SPLINE
SPL {X  -134.058, Y  +288.094, Z    +0.000, E1   +46.503, E3 +177391.868}
SPL {X  -153.979, Y  +327.577, Z    +0.000, E1   +33.452, E3 +177403.408}
SPL {X  -160.130, Y  +351.024, Z    +0.000, E1   +21.715, E3 +177407.838}
SPL {X  -162.127, Y  +365.491, Z    +0.000, E1   +12.692, E3 +177407.762}
SPL {X  -162.801, Y  +378.004, Z    +0.000, E1    +3.811, E3 +177408.178}
SPL {X  -162.820, Y  +382.501, Z    +0.000, E1    +0.028, E3 +177407.596}
SPL {X  -162.820, Y  +385.123, Z    +0.000, E1    -3.284, E3 +177407.274}
SPL {X  -162.820, Y  +390.608, Z    +0.000, E1   -12.198, E3 +177407.187}
SPL {X  -162.820, Y  +396.028, Z    +0.000, E1   -22.022, E3 +177407.055}
SPL {X  -162.820, Y  +402.037, Z    +0.000, E1   -32.247, E3 +177406.993}
SPL {X  -162.820, Y  +411.189, Z    +0.000, E1   -44.140, E3 +177408.323}
SPL {X  -162.820, Y  +422.160, Z    +0.000, E1   -56.042, E3 +177406.794}
SPL {X  -162.820, Y  +475.891, Z    +0.000, E1   -67.666, E3 +177427.113}
SPL {X  -162.820, Y  +573.811, Z    +0.000, E1   -65.269, E3 +177511.711}
SPL {X  -162.820, Y  +580.233, Z    +0.000, E1   -64.427, E3 +177524.418}
SPL {X  -162.820, Y  +590.756, Z    +0.000, E1   -64.410, E3 +177534.986}
SPL {X  -162.820, Y  +600.605, Z    +0.000, E1   -64.446, E3 +177544.559}
SPL {X  -162.820, Y  +611.699, Z    +0.000, E1   -64.369, E3 +177556.238}
SPL {X  -162.820, Y  +622.825, Z    +0.000, E1   -64.446, E3 +177566.683}
SPL {X  -162.820, Y  +635.776, Z    +0.000, E1   -64.495, E3 +177579.372}
SPL {X  -162.820, Y  +648.933, Z    +0.000, E1   -64.417, E3 +177592.920}
SPL {X  -162.820, Y  +658.800, Z    +0.000, E1   -64.418, E3 +177602.734}
SPL {X  -162.820, Y  +670.777, Z    +0.000, E1   -64.432, E3 +177614.647}
SPL {X  -162.296, Y  +686.556, Z    +0.000, E1   -64.388, E3 +177630.850}
SPL {X  -160.469, Y  +701.070, Z    +0.000, E1   -64.058, E3 +177647.753}
SPL {X  -157.811, Y  +713.575, Z    +0.000, E1   -63.758, E3 +177662.332}
SPL {X  -154.601, Y  +724.576, Z    +0.000, E1   -63.303, E3 +177676.454}
SPL {X  -151.802, Y  +732.376, Z    +0.000, E1   -62.761, E3 +177687.581}
SPL {X  -149.758, Y  +737.398, Z    +0.000, E1   -62.434, E3 +177694.602}
SPL {X  -146.903, Y  +743.713, Z    +0.000, E1   -62.188, E3 +177702.375}
SPL {X  -144.901, Y  +747.758, Z    +0.000, E1   -61.566, E3 +177709.838}
SPL {X  -141.375, Y  +754.268, Z    +0.000, E1   -61.208, E3 +177718.391}
SPL {X  -137.988, Y  +759.927, Z    +0.000, E1   -60.537, E3 +177727.190}
SPL {X  -134.516, Y  +765.238, Z    +0.000, E1   -60.629, E3 +177731.993}
SPL {X  -126.113, Y  +776.485, Z    +0.000, E1   -62.672, E3 +177733.554}
SPL {X   -94.739, Y  +805.919, Z    +0.000, E1   -54.063, E3 +177840.294}
ENDSPLINE

SPLINE
SPL {X  -130.051, Y  +771.465, Z    +0.000, E1   -46.832, E3 +177962.078}
SPL {X  -150.288, Y  +736.141, Z    +0.000, E1   -36.889, E3 +177981.934}
SPL {X  -159.122, Y  +708.003, Z    +0.000, E1   -24.018, E3 +177984.643}
SPL {X  -161.938, Y  +690.423, Z    +0.000, E1   -13.625, E3 +177985.854}
SPL {X  -162.746, Y  +678.392, Z    +0.000, E1    -5.513, E3 +177985.927}
SPL {X  -162.820, Y  +672.097, Z    +0.000, E1    -0.584, E3 +177985.631}
SPL {X  -162.820, Y  +670.674, Z    +0.000, E1    +0.808, E3 +177985.263}
SPL {X  -162.820, Y  +666.307, Z    +0.000, E1    +6.851, E3 +177985.046}
SPL {X  -162.820, Y  +660.761, Z    +0.000, E1   +16.102, E3 +177985.188}
SPL {X  -162.820, Y  +655.024, Z    +0.000, E1   +25.730, E3 +177985.350}
SPL {X  -162.820, Y  +646.498, Z    +0.000, E1   +39.738, E3 +177983.871}
SPL {X  -162.820, Y  +637.711, Z    +0.000, E1   +46.793, E3 +177988.363}
SPL {X  -162.820, Y  +598.602, Z    +0.000, E1   +67.541, E3 +177990.914}
SPL {X  -162.820, Y  +578.435, Z    +0.000, E1   +65.472, E3 +178009.014}
SPL {X  -162.820, Y  +475.450, Z    +0.000, E1   +67.130, E3 +178077.952}
ENDSPLINE

SPLINE
SPL {X  -162.820, Y  +483.223, Z    +0.000, E1   +64.312, E3 +178092.391}
SPL {X  -162.820, Y  +502.830, Z    +0.000, E1   +59.229, E3 +178107.312}
ENDSPLINE

SPLINE
SPL {X  -162.820, Y  +486.621, Z    +0.000, E1   +59.661, E3 +178124.231}
SPL {X  -162.820, Y  +472.771, Z    +0.000, E1   +60.369, E3 +178135.977}
SPL {X  -162.820, Y  +460.138, Z    +0.000, E1   +61.014, E3 +178146.296}
SPL {X  -162.820, Y  +448.741, Z    +0.000, E1   +61.510, E3 +178155.811}
SPL {X  -162.820, Y  +430.985, Z    +0.000, E1   +62.533, E3 +178168.244}
SPL {X  -162.820, Y  +413.005, Z    +0.000, E1   +63.234, E3 +178182.234}
SPL {X  -162.820, Y  +396.727, Z    +0.000, E1   +63.972, E3 +178193.586}
SPL {X  -162.756, Y  +375.937, Z    +0.000, E1   +64.914, E3 +178207.195}
SPL {X  -161.353, Y  +358.691, Z    +0.000, E1   +65.588, E3 +178218.419}
SPL {X  -159.475, Y  +347.667, Z    +0.000, E1   +65.889, E3 +178226.300}
SPL {X  -157.043, Y  +337.513, Z    +0.000, E1   +65.541, E3 +178238.378}
SPL {X  -154.736, Y  +329.832, Z    +0.000, E1   +65.034, E3 +178248.824}
SPL {X  -151.631, Y  +321.184, Z    +0.000, E1   +64.776, E3 +178258.669}
SPL {X  -147.832, Y  +312.265, Z    +0.000, E1   +64.201, E3 +178270.478}
SPL {X  -145.264, Y  +306.955, Z    +0.000, E1   +63.555, E3 +178279.084}
SPL {X  -142.454, Y  +301.650, Z    +0.000, E1   +63.360, E3 +178285.088}
SPL {X  -139.696, Y  +296.861, Z    +0.000, E1   +62.910, E3 +178291.856}
SPL {X  -137.330, Y  +293.030, Z    +0.000, E1   +62.290, E3 +178298.481}
SPL {X  -134.245, Y  +288.366, Z    +0.000, E1   +62.031, E3 +178303.962}
SPL {X  -128.642, Y  +280.693, Z    +0.000, E1   +63.351, E3 +178304.956}
SPL {X   -90.696, Y  +245.280, Z    +0.000, E1   +54.124, E3 +178425.644}
ENDSPLINE

SPLINE
SPL {X  -134.058, Y  +288.094, Z    +0.000, E1   +46.503, E3 +178553.158}
SPL {X  -148.633, Y  +314.028, Z    +0.000, E1   +38.752, E3 +178562.047}
SPL {X  -156.325, Y  +334.971, Z    +0.000, E1   +30.037, E3 +178565.814}
SPL {X  -160.130, Y  +351.024, Z    +0.000, E1   +21.715, E3 +178569.128}
SPL {X  -162.127, Y  +365.491, Z    +0.000, E1   +12.692, E3 +178569.052}
SPL {X  -162.801, Y  +378.004, Z    +0.000, E1    +3.811, E3 +178569.468}
SPL {X  -162.820, Y  +382.997, Z    +0.000, E1    -0.389, E3 +178568.792}
SPL {X  -162.820, Y  +387.631, Z    +0.000, E1    -7.169, E3 +178568.551}
SPL {X  -162.820, Y  +394.064, Z    +0.000, E1   -18.298, E3 +178568.361}
SPL {X  -162.820, Y  +402.037, Z    +0.000, E1   -32.247, E3 +178568.283}
SPL {X  -162.820, Y  +414.067, Z    +0.000, E1   -47.235, E3 +178569.709}
SPL {X  -162.820, Y  +424.566, Z    +0.000, E1   -59.255, E3 +178566.374}
SPL {X  -162.820, Y  +460.664, Z    +0.000, E1   -69.605, E3 +178574.671}
SPL {X  -162.820, Y  +481.040, Z    +0.000, E1   -67.047, E3 +178593.259}
SPL {X  -162.820, Y  +573.811, Z    +0.000, E1   -65.269, E3 +178673.001}
SPL {X  -162.820, Y  +580.233, Z    +0.000, E1   -64.427, E3 +178685.708}
SPL {X  -162.820, Y  +590.756, Z    +0.000, E1   -64.410, E3 +178696.276}
SPL {X  -162.820, Y  +600.605, Z    +0.000, E1   -64.446, E3 +178705.849}
SPL {X  -162.820, Y  +611.699, Z    +0.000, E1   -64.369, E3 +178717.529}
SPL {X  -162.820, Y  +622.825, Z    +0.000, E1   -64.446, E3 +178727.973}
SPL {X  -162.820, Y  +635.776, Z    +0.000, E1   -64.495, E3 +178740.663}
SPL {X  -162.820, Y  +648.933, Z    +0.000, E1   -64.417, E3 +178754.210}
SPL {X  -162.820, Y  +658.800, Z    +0.000, E1   -64.418, E3 +178764.024}
SPL {X  -162.820, Y  +670.777, Z    +0.000, E1   -64.432, E3 +178775.937}
SPL {X  -162.296, Y  +686.556, Z    +0.000, E1   -64.388, E3 +178792.140}
SPL {X  -160.469, Y  +701.070, Z    +0.000, E1   -64.058, E3 +178809.044}
SPL {X  -157.811, Y  +713.575, Z    +0.000, E1   -63.758, E3 +178823.622}
SPL {X  -155.696, Y  +721.135, Z    +0.000, E1   -63.387, E3 +178833.556}
SPL {X  -153.915, Y  +726.609, Z    +0.000, E1   -63.196, E3 +178840.330}
SPL {X  -151.802, Y  +732.376, Z    +0.000, E1   -62.761, E3 +178848.872}
SPL {X  -149.758, Y  +737.398, Z    +0.000, E1   -62.434, E3 +178855.892}
SPL {X  -146.903, Y  +743.713, Z    +0.000, E1   -62.188, E3 +178863.665}
SPL {X  -143.515, Y  +750.401, Z    +0.000, E1   -61.484, E3 +178874.349}
SPL {X  -140.303, Y  +756.116, Z    +0.000, E1   -60.974, E3 +178882.547}
SPL {X  -137.124, Y  +761.291, Z    +0.000, E1   -60.398, E3 +178890.593}
SPL {X  -130.896, Y  +770.333, Z    +0.000, E1   -61.755, E3 +178893.268}
SPL {X   -94.739, Y  +805.919, Z    +0.000, E1   -54.063, E3 +179001.585}
ENDSPLINE

SPLINE
SPL {X  -130.051, Y  +771.465, Z    +0.000, E1   -46.832, E3 +179123.369}
SPL {X  -154.243, Y  +725.647, Z    +0.000, E1   -32.659, E3 +179144.931}
SPL {X  -160.324, Y  +701.901, Z    +0.000, E1   -20.534, E3 +179145.754}
SPL {X  -161.938, Y  +690.423, Z    +0.000, E1   -13.625, E3 +179147.144}
SPL {X  -162.638, Y  +681.194, Z    +0.000, E1    -7.430, E3 +179146.965}
SPL {X  -162.820, Y  +672.793, Z    +0.000, E1    -1.263, E3 +179147.023}
SPL {X  -162.820, Y  +670.674, Z    +0.000, E1    +0.808, E3 +179146.553}
SPL {X  -162.820, Y  +666.307, Z    +0.000, E1    +6.851, E3 +179146.336}
SPL {X  -162.820, Y  +660.761, Z    +0.000, E1   +16.102, E3 +179146.479}
SPL {X  -162.820, Y  +655.024, Z    +0.000, E1   +25.730, E3 +179146.640}
SPL {X  -162.820, Y  +646.498, Z    +0.000, E1   +39.738, E3 +179145.161}
SPL {X  -162.820, Y  +637.711, Z    +0.000, E1   +46.793, E3 +179149.653}
SPL {X  -162.820, Y  +598.602, Z    +0.000, E1   +67.541, E3 +179152.204}
SPL {X  -162.820, Y  +578.435, Z    +0.000, E1   +65.472, E3 +179170.304}
SPL {X  -162.820, Y  +475.450, Z    +0.000, E1   +67.130, E3 +179239.242}
ENDSPLINE

SPLINE
SPL {X  -162.820, Y  +483.223, Z    +0.000, E1   +64.312, E3 +179253.681}
SPL {X  -162.820, Y  +502.830, Z    +0.000, E1   +59.229, E3 +179268.602}
ENDSPLINE

SPLINE
SPL {X  -162.820, Y  +486.621, Z    +0.000, E1   +59.661, E3 +179285.522}
SPL {X  -162.820, Y  +472.771, Z    +0.000, E1   +60.369, E3 +179297.267}
SPL {X  -162.820, Y  +460.138, Z    +0.000, E1   +61.014, E3 +179307.587}
SPL {X  -162.820, Y  +448.741, Z    +0.000, E1   +61.510, E3 +179317.102}
SPL {X  -162.820, Y  +430.985, Z    +0.000, E1   +62.533, E3 +179329.535}
SPL {X  -162.820, Y  +413.005, Z    +0.000, E1   +63.234, E3 +179343.525}
SPL {X  -162.820, Y  +396.727, Z    +0.000, E1   +63.972, E3 +179354.876}
SPL {X  -162.820, Y  +382.966, Z    +0.000, E1   +64.511, E3 +179364.598}
SPL {X  -161.867, Y  +362.911, Z    +0.000, E1   +65.480, E3 +179376.672}
SPL {X  -158.833, Y  +344.688, Z    +0.000, E1   +65.800, E3 +179391.172}
SPL {X  -155.590, Y  +332.521, Z    +0.000, E1   +65.288, E3 +179406.106}
SPL {X  -151.631, Y  +321.184, Z    +0.000, E1   +64.776, E3 +179419.959}
SPL {X  -147.832, Y  +312.265, Z    +0.000, E1   +64.201, E3 +179431.769}
SPL {X  -145.264, Y  +306.955, Z    +0.000, E1   +63.555, E3 +179440.375}
SPL {X  -142.454, Y  +301.650, Z    +0.000, E1   +63.360, E3 +179446.378}
SPL {X  -139.696, Y  +296.861, Z    +0.000, E1   +62.910, E3 +179453.146}
SPL {X  -137.330, Y  +293.030, Z    +0.000, E1   +62.290, E3 +179459.771}
SPL {X  -134.245, Y  +288.366, Z    +0.000, E1   +62.031, E3 +179465.252}
SPL {X  -128.642, Y  +280.693, Z    +0.000, E1   +63.351, E3 +179466.246}
SPL {X   -90.696, Y  +245.280, Z    +0.000, E1   +54.124, E3 +179586.935}
ENDSPLINE

SPLINE
SPL {X  -134.058, Y  +288.094, Z    +0.000, E1   +46.503, E3 +179714.448}
SPL {X  -153.979, Y  +327.577, Z    +0.000, E1   +33.452, E3 +179725.988}
SPL {X  -160.130, Y  +351.024, Z    +0.000, E1   +21.715, E3 +179730.419}
SPL {X  -162.127, Y  +365.491, Z    +0.000, E1   +12.692, E3 +179730.342}
SPL {X  -162.801, Y  +378.004, Z    +0.000, E1    +3.811, E3 +179730.758}
SPL {X  -162.820, Y  +382.501, Z    +0.000, E1    +0.028, E3 +179730.177}
SPL {X  -162.820, Y  +385.123, Z    +0.000, E1    -3.284, E3 +179729.854}
SPL {X  -162.820, Y  +390.608, Z    +0.000, E1   -12.198, E3 +179729.768}
SPL {X  -162.820, Y  +396.028, Z    +0.000, E1   -22.022, E3 +179729.636}
SPL {X  -162.820, Y  +402.037, Z    +0.000, E1   -32.247, E3 +179729.573}
SPL {X  -162.820, Y  +411.189, Z    +0.000, E1   -44.140, E3 +179730.903}
SPL {X  -162.820, Y  +422.160, Z    +0.000, E1   -56.042, E3 +179729.375}
SPL {X  -162.820, Y  +475.891, Z    +0.000, E1   -67.666, E3 +179749.694}
SPL {X  -162.820, Y  +573.811, Z    +0.000, E1   -65.269, E3 +179834.292}
SPL {X  -162.820, Y  +580.233, Z    +0.000, E1   -64.427, E3 +179846.999}
SPL {X  -162.820, Y  +590.756, Z    +0.000, E1   -64.410, E3 +179857.566}
SPL {X  -162.820, Y  +600.605, Z    +0.000, E1   -64.446, E3 +179867.139}
SPL {X  -162.820, Y  +611.699, Z    +0.000, E1   -64.369, E3 +179878.819}
SPL {X  -162.820, Y  +625.950, Z    +0.000, E1   -64.427, E3 +179892.659}
SPL {X  -162.820, Y  +639.401, Z    +0.000, E1   -64.540, E3 +179905.082}
SPL {X  -162.820, Y  +648.933, Z    +0.000, E1   -64.417, E3 +179915.500}
SPL {X  -162.820, Y  +658.800, Z    +0.000, E1   -64.418, E3 +179925.314}
SPL {X  -162.820, Y  +670.777, Z    +0.000, E1   -64.432, E3 +179937.228}
SPL {X  -162.296, Y  +686.556, Z    +0.000, E1   -64.388, E3 +179953.431}
SPL {X  -161.171, Y  +696.611, Z    +0.000, E1   -64.029, E3 +179965.896}
SPL {X  -159.311, Y  +707.123, Z    +0.000, E1   -64.022, E3 +179976.590}
SPL {X  -156.625, Y  +717.984, Z    +0.000, E1   -63.524, E3 +179990.944}
SPL {X  -153.915, Y  +726.609, Z    +0.000, E1   -63.196, E3 +180001.621}
SPL {X  -151.802, Y  +732.376, Z    +0.000, E1   -62.761, E3 +180010.162}
SPL {X  -149.758, Y  +737.398, Z    +0.000, E1   -62.434, E3 +180017.182}
SPL {X  -146.903, Y  +743.713, Z    +0.000, E1   -62.188, E3 +180024.955}
SPL {X  -143.515, Y  +750.401, Z    +0.000, E1   -61.484, E3 +180035.639}
SPL {X  -140.303, Y  +756.116, Z    +0.000, E1   -60.974, E3 +180043.837}
SPL {X  -137.124, Y  +761.291, Z    +0.000, E1   -60.398, E3 +180051.884}
SPL {X  -130.896, Y  +770.333, Z    +0.000, E1   -61.755, E3 +180054.558}
SPL {X   -95.040, Y  +805.704, Z    +0.000, E1   -55.103, E3 +180147.094}
ENDSPLINE

SPLINE
SPL {X   -95.634, Y  +805.274, Z    +0.000, E1   -52.767, E3 +180186.253}
SPL {X  -130.051, Y  +771.465, Z    +0.000, E1   -46.832, E3 +180284.659}
SPL {X  -154.243, Y  +725.647, Z    +0.000, E1   -32.659, E3 +180306.221}
SPL {X  -161.394, Y  +695.005, Z    +0.000, E1   -16.571, E3 +180307.926}
SPL {X  -162.638, Y  +681.194, Z    +0.000, E1    -7.430, E3 +180308.255}
SPL {X  -162.820, Y  +672.793, Z    +0.000, E1    -1.263, E3 +180308.314}
SPL {X  -162.820, Y  +670.674, Z    +0.000, E1    +0.808, E3 +180307.844}
SPL {X  -162.820, Y  +666.307, Z    +0.000, E1    +6.851, E3 +180307.626}
SPL {X  -162.820, Y  +660.761, Z    +0.000, E1   +16.102, E3 +180307.769}
SPL {X  -162.820, Y  +655.024, Z    +0.000, E1   +25.730, E3 +180307.930}
SPL {X  -162.820, Y  +646.498, Z    +0.000, E1   +39.738, E3 +180306.451}
SPL {X  -162.820, Y  +637.711, Z    +0.000, E1   +46.793, E3 +180310.944}
SPL {X  -162.820, Y  +598.602, Z    +0.000, E1   +67.541, E3 +180313.495}
SPL {X  -162.820, Y  +578.435, Z    +0.000, E1   +65.472, E3 +180331.595}
SPL {X  -162.820, Y  +475.450, Z    +0.000, E1   +67.130, E3 +180400.532}
ENDSPLINE

SPLINE
SPL {X  -162.820, Y  +483.223, Z    +0.000, E1   +64.312, E3 +180414.972}
SPL {X  -162.820, Y  +504.718, Z    +0.000, E1   +59.258, E3 +180427.195}
ENDSPLINE

SPLINE
SPL {X  -162.820, Y  +492.515, Z    +0.000, E1   +59.352, E3 +180441.661}
SPL {X  -162.820, Y  +476.196, Z    +0.000, E1   +60.204, E3 +180455.694}
SPL {X  -162.820, Y  +460.138, Z    +0.000, E1   +61.014, E3 +180468.877}
SPL {X  -162.820, Y  +448.741, Z    +0.000, E1   +61.510, E3 +180478.392}
SPL {X  -162.820, Y  +430.985, Z    +0.000, E1   +62.533, E3 +180490.825}
SPL {X  -162.820, Y  +413.005, Z    +0.000, E1   +63.234, E3 +180504.815}
SPL {X  -162.820, Y  +396.727, Z    +0.000, E1   +63.972, E3 +180516.166}
SPL {X  -162.756, Y  +375.937, Z    +0.000, E1   +64.914, E3 +180529.776}
SPL {X  -161.353, Y  +358.691, Z    +0.000, E1   +65.588, E3 +180541.000}
SPL {X  -158.833, Y  +344.688, Z    +0.000, E1   +65.800, E3 +180552.463}
SPL {X  -155.590, Y  +332.521, Z    +0.000, E1   +65.288, E3 +180567.396}
SPL {X  -151.631, Y  +321.184, Z    +0.000, E1   +64.776, E3 +180581.249}
SPL {X  -147.832, Y  +312.265, Z    +0.000, E1   +64.201, E3 +180593.059}
SPL {X  -145.264, Y  +306.955, Z    +0.000, E1   +63.555, E3 +180601.665}
SPL {X  -142.454, Y  +301.650, Z    +0.000, E1   +63.360, E3 +180607.669}
SPL {X  -139.696, Y  +296.861, Z    +0.000, E1   +62.910, E3 +180614.436}
SPL {X  -137.330, Y  +293.030, Z    +0.000, E1   +62.290, E3 +180621.061}
SPL {X  -134.245, Y  +288.366, Z    +0.000, E1   +62.031, E3 +180626.543}
SPL {X  -128.642, Y  +280.693, Z    +0.000, E1   +63.351, E3 +180627.536}
SPL {X   -90.696, Y  +245.280, Z    +0.000, E1   +54.124, E3 +180748.225}
ENDSPLINE

SPLINE
SPL {X  -134.058, Y  +288.094, Z    +0.000, E1   +46.503, E3 +180875.739}
SPL {X  -148.633, Y  +314.028, Z    +0.000, E1   +38.752, E3 +180884.627}
SPL {X  -156.325, Y  +334.971, Z    +0.000, E1   +30.037, E3 +180888.395}
SPL {X  -160.130, Y  +351.024, Z    +0.000, E1   +21.715, E3 +180891.709}
SPL {X  -162.127, Y  +365.491, Z    +0.000, E1   +12.692, E3 +180891.633}
SPL {X  -162.801, Y  +378.004, Z    +0.000, E1    +3.811, E3 +180892.049}
SPL {X  -162.820, Y  +382.997, Z    +0.000, E1    -0.389, E3 +180891.372}
SPL {X  -162.820, Y  +387.631, Z    +0.000, E1    -7.169, E3 +180891.132}
SPL {X  -162.820, Y  +394.064, Z    +0.000, E1   -18.298, E3 +180890.942}
SPL {X  -162.820, Y  +402.037, Z    +0.000, E1   -32.247, E3 +180890.864}
SPL {X  -162.820, Y  +414.067, Z    +0.000, E1   -47.235, E3 +180892.290}
SPL {X  -162.820, Y  +424.566, Z    +0.000, E1   -59.255, E3 +180888.955}
SPL {X  -162.820, Y  +460.664, Z    +0.000, E1   -69.605, E3 +180897.251}
SPL {X  -162.820, Y  +481.040, Z    +0.000, E1   -67.047, E3 +180915.840}
SPL {X  -162.820, Y  +573.811, Z    +0.000, E1   -65.269, E3 +180995.582}
SPL {X  -162.820, Y  +580.233, Z    +0.000, E1   -64.427, E3 +181008.289}
SPL {X  -162.820, Y  +590.756, Z    +0.000, E1   -64.410, E3 +181018.856}
SPL {X  -162.820, Y  +600.605, Z    +0.000, E1   -64.446, E3 +181028.430}
SPL {X  -162.820, Y  +611.699, Z    +0.000, E1   -64.369, E3 +181040.109}
SPL {X  -162.820, Y  +625.950, Z    +0.000, E1   -64.427, E3 +181053.950}
SPL {X  -162.820, Y  +639.401, Z    +0.000, E1   -64.540, E3 +181066.372}
SPL {X  -162.820, Y  +648.933, Z    +0.000, E1   -64.417, E3 +181076.790}
SPL {X  -162.820, Y  +658.800, Z    +0.000, E1   -64.418, E3 +181086.605}
SPL {X  -162.820, Y  +670.777, Z    +0.000, E1   -64.432, E3 +181098.518}
SPL {X  -162.613, Y  +681.710, Z    +0.000, E1   -64.310, E3 +181110.282}
SPL {X  -161.587, Y  +693.503, Z    +0.000, E1   -64.259, E3 +181122.636}
SPL {X  -159.311, Y  +707.123, Z    +0.000, E1   -64.022, E3 +181137.880}
SPL {X  -156.625, Y  +717.984, Z    +0.000, E1   -63.524, E3 +181152.235}
SPL {X  -153.915, Y  +726.609, Z    +0.000, E1   -63.196, E3 +181162.911}
SPL {X  -151.802, Y  +732.376, Z    +0.000, E1   -62.761, E3 +181171.452}
SPL {X  -149.758, Y  +737.398, Z    +0.000, E1   -62.434, E3 +181178.473}
SPL {X  -146.903, Y  +743.713, Z    +0.000, E1   -62.188, E3 +181186.246}
SPL {X  -143.515, Y  +750.401, Z    +0.000, E1   -61.484, E3 +181196.930}
SPL {X  -138.985, Y  +758.314, Z    +0.000, E1   -60.770, E3 +181208.489}
SPL {X  -133.449, Y  +766.783, Z    +0.000, E1   -60.899, E3 +181216.109}
SPL {X   -94.739, Y  +805.919, Z    +0.000, E1   -54.063, E3 +181324.165}
ENDSPLINE

SPLINE
SPL {X  -130.051, Y  +771.465, Z    +0.000, E1   -46.832, E3 +181445.949}
SPL {X  -150.288, Y  +736.141, Z    +0.000, E1   -36.889, E3 +181465.805}
SPL {X  -159.122, Y  +708.003, Z    +0.000, E1   -24.018, E3 +181468.514}
SPL {X  -161.938, Y  +690.423, Z    +0.000, E1   -13.625, E3 +181469.725}
SPL {X  -162.638, Y  +681.194, Z    +0.000, E1    -7.430, E3 +181469.546}
SPL {X  -162.805, Y  +675.686, Z    +0.000, E1    -3.400, E3 +181470.021}
SPL {X  -162.820, Y  +671.700, Z    +0.000, E1    -0.272, E3 +181469.363}
SPL {X  -162.820, Y  +668.888, Z    +0.000, E1    +3.063, E3 +181469.060}
SPL {X  -162.820, Y  +664.763, Z    +0.000, E1    +9.526, E3 +181468.720}
SPL {X  -162.820, Y  +659.878, Z    +0.000, E1   +17.497, E3 +181469.125}
SPL {X  -162.820, Y  +650.308, Z    +0.000, E1   +33.487, E3 +181468.538}
SPL {X  -162.820, Y  +637.711, Z    +0.000, E1   +46.793, E3 +181472.234}
SPL {X  -162.820, Y  +598.602, Z    +0.000, E1   +67.541, E3 +181474.785}
SPL {X  -162.820, Y  +578.435, Z    +0.000, E1   +65.472, E3 +181492.885}
SPL {X  -162.820, Y  +475.450, Z    +0.000, E1   +67.130, E3 +181561.822}
ENDSPLINE

SPLINE
SPL {X  -162.820, Y  +483.223, Z    +0.000, E1   +64.312, E3 +181576.262}
SPL {X  -162.820, Y  +502.830, Z    +0.000, E1   +59.229, E3 +181591.183}
ENDSPLINE

SPLINE
SPL {X  -162.820, Y  +486.621, Z    +0.000, E1   +59.661, E3 +181608.102}
SPL {X  -162.820, Y  +472.771, Z    +0.000, E1   +60.369, E3 +181619.848}
SPL {X  -162.820, Y  +460.138, Z    +0.000, E1   +61.014, E3 +181630.167}
SPL {X  -162.820, Y  +448.741, Z    +0.000, E1   +61.510, E3 +181639.682}
SPL {X  -162.820, Y  +430.985, Z    +0.000, E1   +62.533, E3 +181652.115}
SPL {X  -162.820, Y  +413.005, Z    +0.000, E1   +63.234, E3 +181666.105}
SPL {X  -162.820, Y  +396.727, Z    +0.000, E1   +63.972, E3 +181677.456}
SPL {X  -162.756, Y  +375.937, Z    +0.000, E1   +64.914, E3 +181691.066}
SPL {X  -161.353, Y  +358.691, Z    +0.000, E1   +65.588, E3 +181702.290}
SPL {X  -159.475, Y  +347.667, Z    +0.000, E1   +65.889, E3 +181710.171}
SPL {X  -157.043, Y  +337.513, Z    +0.000, E1   +65.541, E3 +181722.249}
SPL {X  -153.776, Y  +326.991, Z    +0.000, E1   +65.023, E3 +181735.489}
SPL {X  -149.992, Y  +317.154, Z    +0.000, E1   +64.515, E3 +181747.953}
SPL {X  -146.026, Y  +308.480, Z    +0.000, E1   +63.813, E3 +181760.195}
SPL {X  -142.454, Y  +301.650, Z    +0.000, E1   +63.360, E3 +181768.959}
SPL {X  -139.696, Y  +296.861, Z    +0.000, E1   +62.910, E3 +181775.727}
SPL {X  -137.330, Y  +293.030, Z    +0.000, E1   +62.290, E3 +181782.352}
SPL {X  -134.245, Y  +288.366, Z    +0.000, E1   +62.031, E3 +181787.833}
SPL {X  -128.642, Y  +280.693, Z    +0.000, E1   +63.351, E3 +181788.827}
SPL {X   -90.696, Y  +245.280, Z    +0.000, E1   +54.124, E3 +181909.515}
ENDSPLINE

SPLINE
SPL {X  -134.058, Y  +288.094, Z    +0.000, E1   +46.503, E3 +182037.029}
SPL {X  -153.979, Y  +327.577, Z    +0.000, E1   +33.452, E3 +182048.569}
SPL {X  -160.130, Y  +351.024, Z    +0.000, E1   +21.715, E3 +182052.999}
SPL {X  -162.127, Y  +365.491, Z    +0.000, E1   +12.692, E3 +182052.923}
SPL {X  -162.745, Y  +375.564, Z    +0.000, E1    +5.577, E3 +182053.533}
SPL {X  -162.820, Y  +382.222, Z    +0.000, E1    +0.380, E3 +182052.806}
SPL {X  -162.820, Y  +385.123, Z    +0.000, E1    -3.284, E3 +182052.435}
SPL {X  -162.820, Y  +390.608, Z    +0.000, E1   -12.198, E3 +182052.348}
SPL {X  -162.820, Y  +396.028, Z    +0.000, E1   -22.022, E3 +182052.216}
SPL {X  -162.820, Y  +402.037, Z    +0.000, E1   -32.247, E3 +182052.154}
SPL {X  -162.820, Y  +414.067, Z    +0.000, E1   -47.235, E3 +182053.580}
SPL {X  -162.820, Y  +424.566, Z    +0.000, E1   -59.255, E3 +182050.245}
SPL {X  -162.820, Y  +460.664, Z    +0.000, E1   -69.605, E3 +182058.542}
SPL {X  -162.820, Y  +481.040, Z    +0.000, E1   -67.047, E3 +182077.130}
SPL {X  -162.820, Y  +573.811, Z    +0.000, E1   -65.269, E3 +182156.872}
SPL {X  -162.820, Y  +580.233, Z    +0.000, E1   -64.427, E3 +182169.579}
SPL {X  -162.820, Y  +590.756, Z    +0.000, E1   -64.410, E3 +182180.147}
SPL {X  -162.820, Y  +600.605, Z    +0.000, E1   -64.446, E3 +182189.720}
SPL {X  -162.820, Y  +611.699, Z    +0.000, E1   -64.369, E3 +182201.400}
SPL {X  -162.820, Y  +622.825, Z    +0.000, E1   -64.446, E3 +182211.844}
SPL {X  -162.820, Y  +635.776, Z    +0.000, E1   -64.495, E3 +182224.534}
SPL {X  -162.820, Y  +648.933, Z    +0.000, E1   -64.417, E3 +182238.081}
SPL {X  -162.820, Y  +658.800, Z    +0.000, E1   -64.418, E3 +182247.895}
SPL {X  -162.820, Y  +670.777, Z    +0.000, E1   -64.432, E3 +182259.808}
SPL {X  -162.296, Y  +686.556, Z    +0.000, E1   -64.388, E3 +182276.011}
SPL {X  -160.469, Y  +701.070, Z    +0.000, E1   -64.058, E3 +182292.915}
SPL {X  -157.811, Y  +713.575, Z    +0.000, E1   -63.758, E3 +182307.493}
SPL {X  -155.696, Y  +721.135, Z    +0.000, E1   -63.387, E3 +182317.427}
SPL {X  -153.915, Y  +726.609, Z    +0.000, E1   -63.196, E3 +182324.201}
SPL {X  -151.802, Y  +732.376, Z    +0.000, E1   -62.761, E3 +182332.743}
SPL {X  -149.758, Y  +737.398, Z    +0.000, E1   -62.434, E3 +182339.763}
SPL {X  -146.903, Y  +743.713, Z    +0.000, E1   -62.188, E3 +182347.536}
SPL {X  -143.515, Y  +750.401, Z    +0.000, E1   -61.484, E3 +182358.220}
SPL {X  -140.303, Y  +756.116, Z    +0.000, E1   -60.974, E3 +182366.418}
SPL {X  -137.124, Y  +761.291, Z    +0.000, E1   -60.398, E3 +182374.464}
SPL {X  -130.896, Y  +770.333, Z    +0.000, E1   -61.755, E3 +182377.139}
SPL {X   -94.739, Y  +805.919, Z    +0.000, E1   -54.063, E3 +182485.456}
ENDSPLINE

SPLINE
SPL {X  -130.051, Y  +771.465, Z    +0.000, E1   -46.832, E3 +182607.240}
SPL {X  -150.288, Y  +736.141, Z    +0.000, E1   -36.889, E3 +182627.096}
SPL {X  -159.122, Y  +708.003, Z    +0.000, E1   -24.018, E3 +182629.804}
SPL {X  -161.938, Y  +690.423, Z    +0.000, E1   -13.625, E3 +182631.015}
SPL {X  -162.638, Y  +681.194, Z    +0.000, E1    -7.430, E3 +182630.836}
SPL {X  -162.805, Y  +675.686, Z    +0.000, E1    -3.400, E3 +182631.312}
SPL {X  -162.820, Y  +671.700, Z    +0.000, E1    -0.272, E3 +182630.653}
SPL {X  -162.820, Y  +669.993, Z    +0.000, E1    +1.755, E3 +182630.320}
SPL {X  -162.820, Y  +666.307, Z    +0.000, E1    +6.851, E3 +182630.207}
SPL {X  -162.820, Y  +659.878, Z    +0.000, E1   +17.497, E3 +182630.415}
SPL {X  -162.820, Y  +650.308, Z    +0.000, E1   +33.487, E3 +182629.828}
SPL {X  -162.820, Y  +637.711, Z    +0.000, E1   +46.793, E3 +182633.524}
SPL {X  -162.820, Y  +613.264, Z    +0.000, E1   +68.325, E3 +182625.723}
SPL {X  -162.820, Y  +583.199, Z    +0.000, E1   +66.160, E3 +182649.213}
SPL {X  -162.820, Y  +480.401, Z    +0.000, E1   +65.660, E3 +182730.104}
ENDSPLINE

SPLINE
SPL {X  -162.820, Y  +490.253, Z    +0.000, E1   +62.754, E3 +182741.867}
SPL {X  -162.820, Y  +503.236, Z    +0.000, E1   +58.858, E3 +182754.220}
ENDSPLINE

SPLINE
SPL {X  -162.820, Y  +486.621, Z    +0.000, E1   +59.661, E3 +182769.393}
SPL {X  -162.820, Y  +472.771, Z    +0.000, E1   +60.369, E3 +182781.138}
SPL {X  -162.820, Y  +460.138, Z    +0.000, E1   +61.014, E3 +182791.458}
SPL {X  -162.820, Y  +448.741, Z    +0.000, E1   +61.510, E3 +182800.972}
SPL {X  -162.820, Y  +430.985, Z    +0.000, E1   +62.533, E3 +182813.406}
SPL {X  -162.820, Y  +413.005, Z    +0.000, E1   +63.234, E3 +182827.396}
SPL {X  -162.820, Y  +396.727, Z    +0.000, E1   +63.972, E3 +182838.747}
SPL {X  -162.756, Y  +375.937, Z    +0.000, E1   +64.914, E3 +182852.356}
SPL {X  -161.353, Y  +358.691, Z    +0.000, E1   +65.588, E3 +182863.581}
SPL {X  -159.475, Y  +347.667, Z    +0.000, E1   +65.889, E3 +182871.461}
SPL {X  -157.043, Y  +337.513, Z    +0.000, E1   +65.541, E3 +182883.539}
SPL {X  -154.736, Y  +329.832, Z    +0.000, E1   +65.034, E3 +182893.985}
SPL {X  -151.631, Y  +321.184, Z    +0.000, E1   +64.776, E3 +182903.830}
SPL {X  -148.818, Y  +314.443, Z    +0.000, E1   +64.320, E3 +182912.777}
SPL {X  -146.026, Y  +308.480, Z    +0.000, E1   +63.813, E3 +182921.486}
SPL {X  -142.454, Y  +301.650, Z    +0.000, E1   +63.360, E3 +182930.249}
SPL {X  -139.696, Y  +296.861, Z    +0.000, E1   +62.910, E3 +182937.017}
SPL {X  -137.330, Y  +293.030, Z    +0.000, E1   +62.290, E3 +182943.642}
SPL {X  -133.474, Y  +287.253, Z    +0.000, E1   +62.192, E3 +182949.381}
SPL {X  -124.928, Y  +276.081, Z    +0.000, E1   +64.269, E3 +182950.088}
SPL {X   -90.696, Y  +245.280, Z    +0.000, E1   +54.124, E3 +183070.806}
ENDSPLINE

SPLINE
SPL {X  -134.058, Y  +288.094, Z    +0.000, E1   +46.503, E3 +183198.319}
SPL {X  -148.633, Y  +314.028, Z    +0.000, E1   +38.752, E3 +183207.208}
SPL {X  -156.325, Y  +334.971, Z    +0.000, E1   +30.037, E3 +183210.976}
SPL {X  -160.130, Y  +351.024, Z    +0.000, E1   +21.715, E3 +183214.290}
SPL {X  -162.127, Y  +365.491, Z    +0.000, E1   +12.692, E3 +183214.213}
SPL {X  -162.745, Y  +375.564, Z    +0.000, E1    +5.577, E3 +183214.824}
SPL {X  -162.820, Y  +382.222, Z    +0.000, E1    +0.380, E3 +183214.096}
SPL {X  -162.820, Y  +384.010, Z    +0.000, E1    -1.878, E3 +183213.759}
SPL {X  -162.820, Y  +386.358, Z    +0.000, E1    -5.320, E3 +183213.688}
SPL {X  -162.820, Y  +390.608, Z    +0.000, E1   -12.198, E3 +183213.639}
SPL {X  -162.820, Y  +396.028, Z    +0.000, E1   -22.022, E3 +183213.507}
SPL {X  -162.820, Y  +402.037, Z    +0.000, E1   -32.247, E3 +183213.444}
SPL {X  -162.820, Y  +411.189, Z    +0.000, E1   -44.140, E3 +183214.774}
SPL {X  -162.820, Y  +422.160, Z    +0.000, E1   -56.042, E3 +183213.246}
SPL {X  -162.820, Y  +475.891, Z    +0.000, E1   -67.666, E3 +183233.565}
SPL {X  -162.820, Y  +573.811, Z    +0.000, E1   -65.269, E3 +183318.163}
SPL {X  -162.820, Y  +580.233, Z    +0.000, E1   -64.427, E3 +183330.870}
SPL {X  -162.820, Y  +590.756, Z    +0.000, E1   -64.410, E3 +183341.437}
SPL {X  -162.820, Y  +600.605, Z    +0.000, E1   -64.446, E3 +183351.010}
SPL {X  -162.820, Y  +611.699, Z    +0.000, E1   -64.369, E3 +183362.690}
SPL {X  -162.820, Y  +622.825, Z    +0.000, E1   -64.446, E3 +183373.134}
SPL {X  -162.820, Y  +635.776, Z    +0.000, E1   -64.495, E3 +183385.824}
SPL {X  -162.820, Y  +648.933, Z    +0.000, E1   -64.417, E3 +183399.371}
SPL {X  -162.820, Y  +658.800, Z    +0.000, E1   -64.418, E3 +183409.185}
SPL {X  -162.820, Y  +670.777, Z    +0.000, E1   -64.432, E3 +183421.099}
SPL {X  -162.613, Y  +681.710, Z    +0.000, E1   -64.310, E3 +183432.863}
SPL {X  -161.587, Y  +693.503, Z    +0.000, E1   -64.259, E3 +183445.217}
SPL {X  -159.311, Y  +707.123, Z    +0.000, E1   -64.022, E3 +183460.461}
SPL {X  -156.625, Y  +717.984, Z    +0.000, E1   -63.524, E3 +183474.815}
SPL {X  -153.915, Y  +726.609, Z    +0.000, E1   -63.196, E3 +183485.492}
SPL {X  -151.802, Y  +732.376, Z    +0.000, E1   -62.761, E3 +183494.033}
SPL {X  -149.758, Y  +737.398, Z    +0.000, E1   -62.434, E3 +183501.053}
SPL {X  -146.903, Y  +743.713, Z    +0.000, E1   -62.188, E3 +183508.826}
SPL {X  -143.515, Y  +750.401, Z    +0.000, E1   -61.484, E3 +183519.510}
SPL {X  -138.985, Y  +758.314, Z    +0.000, E1   -60.770, E3 +183531.070}
SPL {X  -133.449, Y  +766.783, Z    +0.000, E1   -60.899, E3 +183538.689}
SPL {X   -94.739, Y  +805.919, Z    +0.000, E1   -54.063, E3 +183646.746}
ENDSPLINE

SPLINE
SPL {X  -130.051, Y  +771.465, Z    +0.000, E1   -46.832, E3 +183768.530}
SPL {X  -150.288, Y  +736.141, Z    +0.000, E1   -36.889, E3 +183788.386}
SPL {X  -159.122, Y  +708.003, Z    +0.000, E1   -24.018, E3 +183791.095}
SPL {X  -161.938, Y  +690.423, Z    +0.000, E1   -13.625, E3 +183792.305}
SPL {X  -162.638, Y  +681.194, Z    +0.000, E1    -7.430, E3 +183792.126}
SPL {X  -162.805, Y  +675.686, Z    +0.000, E1    -3.400, E3 +183792.602}
SPL {X  -162.820, Y  +671.700, Z    +0.000, E1    -0.272, E3 +183791.944}
SPL {X  -162.820, Y  +668.888, Z    +0.000, E1    +3.063, E3 +183791.641}
SPL {X  -162.820, Y  +664.763, Z    +0.000, E1    +9.526, E3 +183791.301}
SPL {X  -162.820, Y  +659.878, Z    +0.000, E1   +17.497, E3 +183791.705}
SPL {X  -162.820, Y  +650.308, Z    +0.000, E1   +33.487, E3 +183791.119}
SPL {X  -162.820, Y  +637.711, Z    +0.000, E1   +46.793, E3 +183794.815}
SPL {X  -162.820, Y  +598.602, Z    +0.000, E1   +67.541, E3 +183797.366}
SPL {X  -162.820, Y  +578.435, Z    +0.000, E1   +65.472, E3 +183815.465}
SPL {X  -162.820, Y  +475.450, Z    +0.000, E1   +67.130, E3 +183884.403}
ENDSPLINE

SPLINE
SPL {X  -162.820, Y  +483.223, Z    +0.000, E1   +64.312, E3 +183898.843}
SPL {X  -162.820, Y  +502.830, Z    +0.000, E1   +59.229, E3 +183913.764}
ENDSPLINE

SPLINE
SPL {X  -162.820, Y  +486.621, Z    +0.000, E1   +59.661, E3 +183930.683}
SPL {X  -162.820, Y  +472.771, Z    +0.000, E1   +60.369, E3 +183942.428}
SPL {X  -162.820, Y  +460.138, Z    +0.000, E1   +61.014, E3 +183952.748}
SPL {X  -162.820, Y  +448.741, Z    +0.000, E1   +61.510, E3 +183962.263}
SPL {X  -162.820, Y  +430.985, Z    +0.000, E1   +62.533, E3 +183974.696}
SPL {X  -162.820, Y  +413.005, Z    +0.000, E1   +63.234, E3 +183988.686}
SPL {X  -162.820, Y  +396.727, Z    +0.000, E1   +63.972, E3 +184000.037}
SPL {X  -162.756, Y  +375.937, Z    +0.000, E1   +64.914, E3 +184013.647}
SPL {X  -161.353, Y  +358.691, Z    +0.000, E1   +65.588, E3 +184024.871}
SPL {X  -159.475, Y  +347.667, Z    +0.000, E1   +65.889, E3 +184032.752}
SPL {X  -157.043, Y  +337.513, Z    +0.000, E1   +65.541, E3 +184044.830}
SPL {X  -154.736, Y  +329.832, Z    +0.000, E1   +65.034, E3 +184055.276}
SPL {X  -151.631, Y  +321.184, Z    +0.000, E1   +64.776, E3 +184065.120}
SPL {X  -147.832, Y  +312.265, Z    +0.000, E1   +64.201, E3 +184076.930}
SPL {X  -145.264, Y  +306.955, Z    +0.000, E1   +63.555, E3 +184085.536}
SPL {X  -142.454, Y  +301.650, Z    +0.000, E1   +63.360, E3 +184091.540}
SPL {X  -139.696, Y  +296.861, Z    +0.000, E1   +62.910, E3 +184098.307}
SPL {X  -137.330, Y  +293.030, Z    +0.000, E1   +62.290, E3 +184104.932}
SPL {X  -134.245, Y  +288.366, Z    +0.000, E1   +62.031, E3 +184110.414}
SPL {X  -128.642, Y  +280.693, Z    +0.000, E1   +63.351, E3 +184111.407}
SPL {X   -90.696, Y  +245.280, Z    +0.000, E1   +54.124, E3 +184232.096}
ENDSPLINE

SPLINE
SPL {X  -134.058, Y  +288.094, Z    +0.000, E1   +46.503, E3 +184359.610}
SPL {X  -148.633, Y  +314.028, Z    +0.000, E1   +38.752, E3 +184368.498}
SPL {X  -156.325, Y  +334.971, Z    +0.000, E1   +30.037, E3 +184372.266}
SPL {X  -160.130, Y  +351.024, Z    +0.000, E1   +21.715, E3 +184375.580}
SPL {X  -162.127, Y  +365.491, Z    +0.000, E1   +12.692, E3 +184375.504}
SPL {X  -162.801, Y  +378.004, Z    +0.000, E1    +3.811, E3 +184375.920}
SPL {X  -162.820, Y  +382.997, Z    +0.000, E1    -0.389, E3 +184375.243}
SPL {X  -162.820, Y  +387.631, Z    +0.000, E1    -7.169, E3 +184375.003}
SPL {X  -162.820, Y  +394.064, Z    +0.000, E1   -18.298, E3 +184374.813}
SPL {X  -162.820, Y  +402.037, Z    +0.000, E1   -32.247, E3 +184374.735}
SPL {X  -162.820, Y  +414.067, Z    +0.000, E1   -47.235, E3 +184376.161}
SPL {X  -162.820, Y  +424.566, Z    +0.000, E1   -59.255, E3 +184372.826}
SPL {X  -162.820, Y  +460.664, Z    +0.000, E1   -69.605, E3 +184381.122}
SPL {X  -162.820, Y  +481.040, Z    +0.000, E1   -67.047, E3 +184399.711}
SPL {X  -162.820, Y  +573.811, Z    +0.000, E1   -65.269, E3 +184479.453}
SPL {X  -162.820, Y  +580.233, Z    +0.000, E1   -64.427, E3 +184492.160}
SPL {X  -162.820, Y  +590.756, Z    +0.000, E1   -64.410, E3 +184502.727}
SPL {X  -162.820, Y  +600.605, Z    +0.000, E1   -64.446, E3 +184512.301}
SPL {X  -162.820, Y  +611.699, Z    +0.000, E1   -64.369, E3 +184523.980}
SPL {X  -162.820, Y  +622.825, Z    +0.000, E1   -64.446, E3 +184534.425}
SPL {X  -162.820, Y  +635.776, Z    +0.000, E1   -64.495, E3 +184547.114}
SPL {X  -162.820, Y  +648.933, Z    +0.000, E1   -64.417, E3 +184560.661}
SPL {X  -162.820, Y  +658.800, Z    +0.000, E1   -64.418, E3 +184570.476}
SPL {X  -162.820, Y  +670.777, Z    +0.000, E1   -64.432, E3 +184582.389}
SPL {X  -162.296, Y  +686.556, Z    +0.000, E1   -64.388, E3 +184598.592}
SPL {X  -160.469, Y  +701.070, Z    +0.000, E1   -64.058, E3 +184615.495}
SPL {X  -157.811, Y  +713.575, Z    +0.000, E1   -63.758, E3 +184630.074}
SPL {X  -155.696, Y  +721.135, Z    +0.000, E1   -63.387, E3 +184640.007}
SPL {X  -153.915, Y  +726.609, Z    +0.000, E1   -63.196, E3 +184646.782}
SPL {X  -151.802, Y  +732.376, Z    +0.000, E1   -62.761, E3 +184655.323}
SPL {X  -149.758, Y  +737.398, Z    +0.000, E1   -62.434, E3 +184662.344}
SPL {X  -146.903, Y  +743.713, Z    +0.000, E1   -62.188, E3 +184670.117}
SPL {X  -143.515, Y  +750.401, Z    +0.000, E1   -61.484, E3 +184680.801}
SPL {X  -140.303, Y  +756.116, Z    +0.000, E1   -60.974, E3 +184688.998}
SPL {X  -137.124, Y  +761.291, Z    +0.000, E1   -60.398, E3 +184697.045}
SPL {X  -130.896, Y  +770.333, Z    +0.000, E1   -61.755, E3 +184699.719}
SPL {X   -94.739, Y  +805.919, Z    +0.000, E1   -54.063, E3 +184808.036}
ENDSPLINE

SPLINE
SPL {X  -130.051, Y  +771.465, Z    +0.000, E1   -46.832, E3 +184929.820}
SPL {X  -154.243, Y  +725.647, Z    +0.000, E1   -32.659, E3 +184951.383}
SPL {X  -161.394, Y  +695.005, Z    +0.000, E1   -16.571, E3 +184953.087}
SPL {X  -162.746, Y  +678.392, Z    +0.000, E1    -5.513, E3 +184953.668}
SPL {X  -162.820, Y  +671.128, Z    +0.000, E1    +0.178, E3 +184953.122}
SPL {X  -162.820, Y  +666.307, Z    +0.000, E1    +6.851, E3 +184952.787}
SPL {X  -162.820, Y  +660.761, Z    +0.000, E1   +16.102, E3 +184952.930}
SPL {X  -162.820, Y  +655.024, Z    +0.000, E1   +25.730, E3 +184953.092}
SPL {X  -162.820, Y  +646.498, Z    +0.000, E1   +39.738, E3 +184951.612}
SPL {X  -162.820, Y  +637.711, Z    +0.000, E1   +46.793, E3 +184956.105}
SPL {X  -162.820, Y  +613.264, Z    +0.000, E1   +68.325, E3 +184948.303}
SPL {X  -162.820, Y  +583.199, Z    +0.000, E1   +66.160, E3 +184971.794}
SPL {X  -162.820, Y  +475.450, Z    +0.000, E1   +67.130, E3 +185045.693}
ENDSPLINE

SPLINE
SPL {X  -162.820, Y  +483.223, Z    +0.000, E1   +64.312, E3 +185060.133}
SPL {X  -162.820, Y  +501.391, Z    +0.000, E1   +60.597, E3 +185066.862}
SPL {X  -162.820, Y  +505.887, Z    +0.000, E1   +58.743, E3 +185074.138}
ENDSPLINE

SPLINE
SPL {X  -162.820, Y  +492.515, Z    +0.000, E1   +59.352, E3 +185086.823}
SPL {X  -162.820, Y  +476.196, Z    +0.000, E1   +60.204, E3 +185100.856}
SPL {X  -162.820, Y  +460.138, Z    +0.000, E1   +61.014, E3 +185114.038}
SPL {X  -162.820, Y  +448.741, Z    +0.000, E1   +61.510, E3 +185123.553}
SPL {X  -162.820, Y  +430.985, Z    +0.000, E1   +62.533, E3 +185135.986}
SPL {X  -162.820, Y  +413.005, Z    +0.000, E1   +63.234, E3 +185149.976}
SPL {X  -162.820, Y  +396.727, Z    +0.000, E1   +63.972, E3 +185161.327}
SPL {X  -162.820, Y  +382.966, Z    +0.000, E1   +64.511, E3 +185171.050}
SPL {X  -161.867, Y  +362.911, Z    +0.000, E1   +65.480, E3 +185183.123}
SPL {X  -158.833, Y  +344.688, Z    +0.000, E1   +65.800, E3 +185197.624}
SPL {X  -156.326, Y  +334.977, Z    +0.000, E1   +65.428, E3 +185209.097}
SPL {X  -153.776, Y  +326.991, Z    +0.000, E1   +65.023, E3 +185219.360}
SPL {X  -149.992, Y  +317.154, Z    +0.000, E1   +64.515, E3 +185231.824}
SPL {X  -146.026, Y  +308.480, Z    +0.000, E1   +63.813, E3 +185244.066}
SPL {X  -142.454, Y  +301.650, Z    +0.000, E1   +63.360, E3 +185252.830}
SPL {X  -139.696, Y  +296.861, Z    +0.000, E1   +62.910, E3 +185259.598}
SPL {X  -137.330, Y  +293.030, Z    +0.000, E1   +62.290, E3 +185266.223}
SPL {X  -134.245, Y  +288.366, Z    +0.000, E1   +62.031, E3 +185271.704}
SPL {X  -128.642, Y  +280.693, Z    +0.000, E1   +63.351, E3 +185272.698}
SPL {X   -90.696, Y  +245.280, Z    +0.000, E1   +54.124, E3 +185393.386}
ENDSPLINE

SPLINE
SPL {X  -134.058, Y  +288.094, Z    +0.000, E1   +46.503, E3 +185520.900}
SPL {X  -153.979, Y  +327.577, Z    +0.000, E1   +33.452, E3 +185532.440}
SPL {X  -160.130, Y  +351.024, Z    +0.000, E1   +21.715, E3 +185536.870}
SPL {X  -162.127, Y  +365.491, Z    +0.000, E1   +12.692, E3 +185536.794}
SPL {X  -162.745, Y  +375.564, Z    +0.000, E1    +5.577, E3 +185537.404}
SPL {X  -162.820, Y  +382.222, Z    +0.000, E1    +0.380, E3 +185536.677}
SPL {X  -162.820, Y  +385.123, Z    +0.000, E1    -3.284, E3 +185536.306}
SPL {X  -162.820, Y  +390.608, Z    +0.000, E1   -12.198, E3 +185536.219}
SPL {X  -162.820, Y  +396.028, Z    +0.000, E1   -22.022, E3 +185536.087}
SPL {X  -162.820, Y  +402.037, Z    +0.000, E1   -32.247, E3 +185536.025}
SPL {X  -162.820, Y  +414.067, Z    +0.000, E1   -47.235, E3 +185537.451}
SPL {X  -162.820, Y  +424.566, Z    +0.000, E1   -59.255, E3 +185534.116}
SPL {X  -162.820, Y  +460.664, Z    +0.000, E1   -69.605, E3 +185542.413}
SPL {X  -162.820, Y  +481.040, Z    +0.000, E1   -67.047, E3 +185561.001}
SPL {X  -162.820, Y  +573.811, Z    +0.000, E1   -65.269, E3 +185640.743}
SPL {X  -162.820, Y  +580.233, Z    +0.000, E1   -64.427, E3 +185653.450}
SPL {X  -162.820, Y  +590.756, Z    +0.000, E1   -64.410, E3 +185664.018}
SPL {X  -162.820, Y  +600.605, Z    +0.000, E1   -64.446, E3 +185673.591}
SPL {X  -162.820, Y  +611.699, Z    +0.000, E1   -64.369, E3 +185685.271}
SPL {X  -162.820, Y  +625.950, Z    +0.000, E1   -64.427, E3 +185699.111}
SPL {X  -162.820, Y  +639.401, Z    +0.000, E1   -64.540, E3 +185711.533}
SPL {X  -162.820, Y  +648.933, Z    +0.000, E1   -64.417, E3 +185721.952}
SPL {X  -162.820, Y  +658.800, Z    +0.000, E1   -64.418, E3 +185731.766}
SPL {X  -162.820, Y  +670.777, Z    +0.000, E1   -64.432, E3 +185743.679}
SPL {X  -162.296, Y  +686.556, Z    +0.000, E1   -64.388, E3 +185759.882}
SPL {X  -160.469, Y  +701.070, Z    +0.000, E1   -64.058, E3 +185776.786}
SPL {X  -157.811, Y  +713.575, Z    +0.000, E1   -63.758, E3 +185791.364}
SPL {X  -154.601, Y  +724.576, Z    +0.000, E1   -63.303, E3 +185805.486}
SPL {X  -151.802, Y  +732.376, Z    +0.000, E1   -62.761, E3 +185816.614}
SPL {X  -149.758, Y  +737.398, Z    +0.000, E1   -62.434, E3 +185823.634}
SPL {X  -146.903, Y  +743.713, Z    +0.000, E1   -62.188, E3 +185831.407}
SPL {X  -143.515, Y  +750.401, Z    +0.000, E1   -61.484, E3 +185842.091}
SPL {X  -138.985, Y  +758.314, Z    +0.000, E1   -60.770, E3 +185853.650}
SPL {X  -133.449, Y  +766.783, Z    +0.000, E1   -60.899, E3 +185861.270}
SPL {X   -94.739, Y  +805.919, Z    +0.000, E1   -54.063, E3 +185969.327}
ENDSPLINE

SPLINE
SPL {X  -130.051, Y  +771.465, Z    +0.000, E1   -46.832, E3 +186091.111}
SPL {X  -154.243, Y  +725.647, Z    +0.000, E1   -32.659, E3 +186112.673}
SPL {X  -160.324, Y  +701.901, Z    +0.000, E1   -20.534, E3 +186113.496}
SPL {X  -161.938, Y  +690.423, Z    +0.000, E1   -13.625, E3 +186114.886}
SPL {X  -162.638, Y  +681.194, Z    +0.000, E1    -7.430, E3 +186114.707}
SPL {X  -162.820, Y  +672.793, Z    +0.000, E1    -1.263, E3 +186114.765}
SPL {X  -162.820, Y  +670.674, Z    +0.000, E1    +0.808, E3 +186114.295}
SPL {X  -162.820, Y  +666.307, Z    +0.000, E1    +6.851, E3 +186114.078}
SPL {X  -162.820, Y  +660.761, Z    +0.000, E1   +16.102, E3 +186114.221}
SPL {X  -162.820, Y  +655.024, Z    +0.000, E1   +25.730, E3 +186114.382}
SPL {X  -162.820, Y  +646.498, Z    +0.000, E1   +39.738, E3 +186112.903}
SPL {X  -162.820, Y  +637.711, Z    +0.000, E1   +46.793, E3 +186117.395}
SPL {X  -162.820, Y  +598.602, Z    +0.000, E1   +67.541, E3 +186119.946}
SPL {X  -162.820, Y  +578.435, Z    +0.000, E1   +65.472, E3 +186138.046}
SPL {X  -162.820, Y  +480.401, Z    +0.000, E1   +65.660, E3 +186213.975}
ENDSPLINE

SPLINE
SPL {X  -162.820, Y  +490.253, Z    +0.000, E1   +62.754, E3 +186225.738}
SPL {X  -162.820, Y  +503.236, Z    +0.000, E1   +58.858, E3 +186238.091}
ENDSPLINE

SPLINE
SPL {X  -162.820, Y  +486.621, Z    +0.000, E1   +59.661, E3 +186253.264}
SPL {X  -162.820, Y  +472.771, Z    +0.000, E1   +60.369, E3 +186265.009}
SPL {X  -162.820, Y  +460.138, Z    +0.000, E1   +61.014, E3 +186275.329}
SPL {X  -162.820, Y  +448.741, Z    +0.000, E1   +61.510, E3 +186284.843}
SPL {X  -162.820, Y  +430.985, Z    +0.000, E1   +62.533, E3 +186297.277}
SPL {X  -162.820, Y  +413.005, Z    +0.000, E1   +63.234, E3 +186311.266}
SPL {X  -162.820, Y  +396.727, Z    +0.000, E1   +63.972, E3 +186322.618}
SPL {X  -162.756, Y  +375.937, Z    +0.000, E1   +64.914, E3 +186336.227}
SPL {X  -161.353, Y  +358.691, Z    +0.000, E1   +65.588, E3 +186347.452}
SPL {X  -159.475, Y  +347.667, Z    +0.000, E1   +65.889, E3 +186355.332}
SPL {X  -157.043, Y  +337.513, Z    +0.000, E1   +65.541, E3 +186367.410}
SPL {X  -154.736, Y  +329.832, Z    +0.000, E1   +65.034, E3 +186377.856}
SPL {X  -151.631, Y  +321.184, Z    +0.000, E1   +64.776, E3 +186387.701}
SPL {X  -147.832, Y  +312.265, Z    +0.000, E1   +64.201, E3 +186399.511}
SPL {X  -145.264, Y  +306.955, Z    +0.000, E1   +63.555, E3 +186408.117}
SPL {X  -142.454, Y  +301.650, Z    +0.000, E1   +63.360, E3 +186414.120}
SPL {X  -139.696, Y  +296.861, Z    +0.000, E1   +62.910, E3 +186420.888}
SPL {X  -137.330, Y  +293.030, Z    +0.000, E1   +62.290, E3 +186427.513}
SPL {X  -134.245, Y  +288.366, Z    +0.000, E1   +62.031, E3 +186432.994}
SPL {X  -128.642, Y  +280.693, Z    +0.000, E1   +63.351, E3 +186433.988}
SPL {X   -90.696, Y  +245.280, Z    +0.000, E1   +54.124, E3 +186554.677}
ENDSPLINE

SPLINE
SPL {X  -134.058, Y  +288.094, Z    +0.000, E1   +46.503, E3 +186682.190}
SPL {X  -153.979, Y  +327.577, Z    +0.000, E1   +33.452, E3 +186693.730}
SPL {X  -160.130, Y  +351.024, Z    +0.000, E1   +21.715, E3 +186698.161}
SPL {X  -162.127, Y  +365.491, Z    +0.000, E1   +12.692, E3 +186698.084}
SPL {X  -162.745, Y  +375.564, Z    +0.000, E1    +5.577, E3 +186698.695}
SPL {X  -162.820, Y  +382.222, Z    +0.000, E1    +0.380, E3 +186697.967}
SPL {X  -162.820, Y  +384.010, Z    +0.000, E1    -1.878, E3 +186697.630}
SPL {X  -162.820, Y  +387.631, Z    +0.000, E1    -7.169, E3 +186697.583}
SPL {X  -162.820, Y  +394.064, Z    +0.000, E1   -18.298, E3 +186697.394}
SPL {X  -162.820, Y  +402.037, Z    +0.000, E1   -32.247, E3 +186697.315}
SPL {X  -162.820, Y  +411.189, Z    +0.000, E1   -44.140, E3 +186698.645}
SPL {X  -162.820, Y  +422.160, Z    +0.000, E1   -56.042, E3 +186697.117}
SPL {X  -162.820, Y  +475.891, Z    +0.000, E1   -67.666, E3 +186717.435}
SPL {X  -162.820, Y  +573.811, Z    +0.000, E1   -65.269, E3 +186802.034}
SPL {X  -162.820, Y  +580.233, Z    +0.000, E1   -64.427, E3 +186814.740}
SPL {X  -162.820, Y  +590.756, Z    +0.000, E1   -64.410, E3 +186825.308}
SPL {X  -162.820, Y  +600.605, Z    +0.000, E1   -64.446, E3 +186834.881}
SPL {X  -162.820, Y  +611.699, Z    +0.000, E1   -64.369, E3 +186846.561}
SPL {X  -162.820, Y  +622.825, Z    +0.000, E1   -64.446, E3 +186857.005}
SPL {X  -162.820, Y  +635.776, Z    +0.000, E1   -64.495, E3 +186869.695}
SPL {X  -162.820, Y  +648.933, Z    +0.000, E1   -64.417, E3 +186883.242}
SPL {X  -162.820, Y  +658.800, Z    +0.000, E1   -64.418, E3 +186893.056}
SPL {X  -162.820, Y  +670.777, Z    +0.000, E1   -64.432, E3 +186904.970}
SPL {X  -162.296, Y  +686.556, Z    +0.000, E1   -64.388, E3 +186921.173}
SPL {X  -160.469, Y  +701.070, Z    +0.000, E1   -64.058, E3 +186938.076}
SPL {X  -157.811, Y  +713.575, Z    +0.000, E1   -63.758, E3 +186952.655}
SPL {X  -155.696, Y  +721.135, Z    +0.000, E1   -63.387, E3 +186962.588}
SPL {X  -153.915, Y  +726.609, Z    +0.000, E1   -63.196, E3 +186969.363}
SPL {X  -151.802, Y  +732.376, Z    +0.000, E1   -62.761, E3 +186977.904}
SPL {X  -149.758, Y  +737.398, Z    +0.000, E1   -62.434, E3 +186984.924}
SPL {X  -146.903, Y  +743.713, Z    +0.000, E1   -62.188, E3 +186992.697}
SPL {X  -144.901, Y  +747.758, Z    +0.000, E1   -61.566, E3 +187000.160}
SPL {X  -141.375, Y  +754.268, Z    +0.000, E1   -61.208, E3 +187008.714}
SPL {X  -137.124, Y  +761.291, Z    +0.000, E1   -60.398, E3 +187019.626}
SPL {X  -130.896, Y  +770.333, Z    +0.000, E1   -61.755, E3 +187022.300}
SPL {X   -94.739, Y  +805.919, Z    +0.000, E1   -54.063, E3 +187130.617}
ENDSPLINE

SPLINE
SPL {X  -130.051, Y  +771.465, Z    +0.000, E1   -46.832, E3 +187252.401}
SPL {X  -150.288, Y  +736.141, Z    +0.000, E1   -36.889, E3 +187272.257}
SPL {X  -159.122, Y  +708.003, Z    +0.000, E1   -24.018, E3 +187274.966}
SPL {X  -161.938, Y  +690.423, Z    +0.000, E1   -13.625, E3 +187276.176}
SPL {X  -162.746, Y  +678.392, Z    +0.000, E1    -5.513, E3 +187276.249}
SPL {X  -162.820, Y  +671.700, Z    +0.000, E1    -0.272, E3 +187275.815}
SPL {X  -162.820, Y  +668.888, Z    +0.000, E1    +3.063, E3 +187275.512}
SPL {X  -162.820, Y  +664.763, Z    +0.000, E1    +9.526, E3 +187275.172}
SPL {X  -162.820, Y  +660.761, Z    +0.000, E1   +16.102, E3 +187275.511}
SPL {X  -162.820, Y  +655.024, Z    +0.000, E1   +25.730, E3 +187275.672}
SPL {X  -162.820, Y  +646.498, Z    +0.000, E1   +39.738, E3 +187274.193}
SPL {X  -162.820, Y  +637.711, Z    +0.000, E1   +46.793, E3 +187278.686}
SPL {X  -162.820, Y  +613.264, Z    +0.000, E1   +68.325, E3 +187270.884}
SPL {X  -162.820, Y  +583.199, Z    +0.000, E1   +66.160, E3 +187294.374}
SPL {X  -162.820, Y  +480.401, Z    +0.000, E1   +65.660, E3 +187375.266}
ENDSPLINE

SPLINE
SPL {X  -162.820, Y  +490.253, Z    +0.000, E1   +62.754, E3 +187387.028}
SPL {X  -162.820, Y  +503.236, Z    +0.000, E1   +58.858, E3 +187399.382}
ENDSPLINE

SPLINE
SPL {X  -162.820, Y  +486.621, Z    +0.000, E1   +59.661, E3 +187414.554}
SPL {X  -162.820, Y  +472.771, Z    +0.000, E1   +60.369, E3 +187426.299}
SPL {X  -162.820, Y  +460.138, Z    +0.000, E1   +61.014, E3 +187436.619}
SPL {X  -162.820, Y  +448.741, Z    +0.000, E1   +61.510, E3 +187446.134}
SPL {X  -162.820, Y  +430.985, Z    +0.000, E1   +62.533, E3 +187458.567}
SPL {X  -162.820, Y  +413.005, Z    +0.000, E1   +63.234, E3 +187472.557}
SPL {X  -162.820, Y  +396.727, Z    +0.000, E1   +63.972, E3 +187483.908}
SPL {X  -162.756, Y  +375.937, Z    +0.000, E1   +64.914, E3 +187497.517}
SPL {X  -161.353, Y  +358.691, Z    +0.000, E1   +65.588, E3 +187508.742}
SPL {X  -159.475, Y  +347.667, Z    +0.000, E1   +65.889, E3 +187516.623}
SPL {X  -157.043, Y  +337.513, Z    +0.000, E1   +65.541, E3 +187528.701}
SPL {X  -153.776, Y  +326.991, Z    +0.000, E1   +65.023, E3 +187541.941}
SPL {X  -149.992, Y  +317.154, Z    +0.000, E1   +64.515, E3 +187554.405}
SPL {X  -146.026, Y  +308.480, Z    +0.000, E1   +63.813, E3 +187566.647}
SPL {X  -142.454, Y  +301.650, Z    +0.000, E1   +63.360, E3 +187575.411}
SPL {X  -139.696, Y  +296.861, Z    +0.000, E1   +62.910, E3 +187582.178}
SPL {X  -137.330, Y  +293.030, Z    +0.000, E1   +62.290, E3 +187588.803}
SPL {X  -134.245, Y  +288.366, Z    +0.000, E1   +62.031, E3 +187594.285}
SPL {X  -128.642, Y  +280.693, Z    +0.000, E1   +63.351, E3 +187595.278}
SPL {X   -90.696, Y  +245.280, Z    +0.000, E1   +54.124, E3 +187715.967}
ENDSPLINE

SPLINE
SPL {X  -134.058, Y  +288.094, Z    +0.000, E1   +46.503, E3 +187843.481}
SPL {X  -148.633, Y  +314.028, Z    +0.000, E1   +38.752, E3 +187852.369}
SPL {X  -156.325, Y  +334.971, Z    +0.000, E1   +30.037, E3 +187856.137}
SPL {X  -160.130, Y  +351.024, Z    +0.000, E1   +21.715, E3 +187859.451}
SPL {X  -162.127, Y  +365.491, Z    +0.000, E1   +12.692, E3 +187859.375}
SPL {X  -162.801, Y  +378.004, Z    +0.000, E1    +3.811, E3 +187859.791}
SPL {X  -162.820, Y  +382.997, Z    +0.000, E1    -0.389, E3 +187859.114}
SPL {X  -162.820, Y  +386.358, Z    +0.000, E1    -5.320, E3 +187858.849}
SPL {X  -162.820, Y  +390.608, Z    +0.000, E1   -12.198, E3 +187858.800}
SPL {X  -162.820, Y  +396.028, Z    +0.000, E1   -22.022, E3 +187858.668}
SPL {X  -162.820, Y  +402.037, Z    +0.000, E1   -32.247, E3 +187858.606}
SPL {X  -162.820, Y  +411.189, Z    +0.000, E1   -44.140, E3 +187859.936}
SPL {X  -162.820, Y  +422.160, Z    +0.000, E1   -56.042, E3 +187858.407}
SPL {X  -162.820, Y  +475.891, Z    +0.000, E1   -67.666, E3 +187878.726}
SPL {X  -162.820, Y  +576.352, Z    +0.000, E1   -67.140, E3 +187951.100}
ENDSPLINE

SPLINE
SPL {X  -162.820, Y  +573.336, Z    +0.000, E1   -64.995, E3 +187964.853}
ENDSPLINE

SPLINE
SPL {X  -162.820, Y  +580.233, Z    +0.000, E1   -64.427, E3 +187976.031}
SPL {X  -162.820, Y  +590.756, Z    +0.000, E1   -64.410, E3 +187986.598}
SPL {X  -162.820, Y  +600.605, Z    +0.000, E1   -64.446, E3 +187996.172}
SPL {X  -162.820, Y  +611.699, Z    +0.000, E1   -64.369, E3 +188007.851}
SPL {X  -162.820, Y  +625.950, Z    +0.000, E1   -64.427, E3 +188021.691}
SPL {X  -162.820, Y  +639.401, Z    +0.000, E1   -64.540, E3 +188034.114}
SPL {X  -162.820, Y  +648.933, Z    +0.000, E1   -64.417, E3 +188044.532}
SPL {X  -162.820, Y  +658.800, Z    +0.000, E1   -64.418, E3 +188054.347}
SPL {X  -162.820, Y  +670.777, Z    +0.000, E1   -64.432, E3 +188066.260}
SPL {X  -162.296, Y  +686.556, Z    +0.000, E1   -64.388, E3 +188082.463}
SPL {X  -161.171, Y  +696.611, Z    +0.000, E1   -64.029, E3 +188094.928}
SPL {X  -159.311, Y  +707.123, Z    +0.000, E1   -64.022, E3 +188105.622}
SPL {X  -156.625, Y  +717.984, Z    +0.000, E1   -63.524, E3 +188119.977}
SPL {X  -153.915, Y  +726.609, Z    +0.000, E1   -63.196, E3 +188130.653}
SPL {X  -151.802, Y  +732.376, Z    +0.000, E1   -62.761, E3 +188139.194}
SPL {X  -149.758, Y  +737.398, Z    +0.000, E1   -62.434, E3 +188146.215}
SPL {X  -146.903, Y  +743.713, Z    +0.000, E1   -62.188, E3 +188153.987}
SPL {X  -143.515, Y  +750.401, Z    +0.000, E1   -61.484, E3 +188164.672}
SPL {X  -140.303, Y  +756.116, Z    +0.000, E1   -60.974, E3 +188172.869}
SPL {X  -137.124, Y  +761.291, Z    +0.000, E1   -60.398, E3 +188180.916}
SPL {X  -130.896, Y  +770.333, Z    +0.000, E1   -61.755, E3 +188183.590}
SPL {X   -94.739, Y  +805.919, Z    +0.000, E1   -54.063, E3 +188291.907}
ENDSPLINE

SPLINE
SPL {X  -130.051, Y  +771.465, Z    +0.000, E1   -46.832, E3 +188413.691}
SPL {X  -154.243, Y  +725.647, Z    +0.000, E1   -32.659, E3 +188435.254}
SPL {X  -161.394, Y  +695.005, Z    +0.000, E1   -16.571, E3 +188436.958}
SPL {X  -162.746, Y  +678.392, Z    +0.000, E1    -5.513, E3 +188437.539}
SPL {X  -162.820, Y  +671.700, Z    +0.000, E1    -0.272, E3 +188437.105}
SPL {X  -162.820, Y  +668.888, Z    +0.000, E1    +3.063, E3 +188436.802}
SPL {X  -162.820, Y  +664.763, Z    +0.000, E1    +9.526, E3 +188436.462}
SPL {X  -162.820, Y  +660.761, Z    +0.000, E1   +16.102, E3 +188436.801}
SPL {X  -162.820, Y  +655.024, Z    +0.000, E1   +25.730, E3 +188436.963}
SPL {X  -162.820, Y  +646.498, Z    +0.000, E1   +39.738, E3 +188435.483}
SPL {X  -162.820, Y  +637.711, Z    +0.000, E1   +46.793, E3 +188439.976}
SPL {X  -162.820, Y  +598.602, Z    +0.000, E1   +67.541, E3 +188442.527}
SPL {X  -162.820, Y  +578.435, Z    +0.000, E1   +65.472, E3 +188460.627}
SPL {X  -162.820, Y  +475.450, Z    +0.000, E1   +67.130, E3 +188529.564}
ENDSPLINE

SPLINE
SPL {X  -162.820, Y  +483.223, Z    +0.000, E1   +64.312, E3 +188544.004}
SPL {X  -162.820, Y  +502.830, Z    +0.000, E1   +59.229, E3 +188558.925}
ENDSPLINE

SPLINE
SPL {X  -162.820, Y  +486.621, Z    +0.000, E1   +59.661, E3 +188575.844}
SPL {X  -162.820, Y  +472.771, Z    +0.000, E1   +60.369, E3 +188587.590}
SPL {X  -162.820, Y  +460.138, Z    +0.000, E1   +61.014, E3 +188597.909}
SPL {X  -162.820, Y  +448.741, Z    +0.000, E1   +61.510, E3 +188607.424}
SPL {X  -162.820, Y  +430.985, Z    +0.000, E1   +62.533, E3 +188619.857}
SPL {X  -162.820, Y  +413.005, Z    +0.000, E1   +63.234, E3 +188633.847}
SPL {X  -162.820, Y  +396.727, Z    +0.000, E1   +63.972, E3 +188645.198}
SPL {X  -162.820, Y  +382.966, Z    +0.000, E1   +64.511, E3 +188654.921}
SPL {X  -161.867, Y  +362.911, Z    +0.000, E1   +65.480, E3 +188666.994}
SPL {X  -159.475, Y  +347.667, Z    +0.000, E1   +65.889, E3 +188677.913}
SPL {X  -157.043, Y  +337.513, Z    +0.000, E1   +65.541, E3 +188689.991}
SPL {X  -153.776, Y  +326.991, Z    +0.000, E1   +65.023, E3 +188703.231}
SPL {X  -150.991, Y  +319.573, Z    +0.000, E1   +64.614, E3 +188712.685}
SPL {X  -147.832, Y  +312.265, Z    +0.000, E1   +64.201, E3 +188722.091}
SPL {X  -145.264, Y  +306.955, Z    +0.000, E1   +63.555, E3 +188730.697}
SPL {X  -142.454, Y  +301.650, Z    +0.000, E1   +63.360, E3 +188736.701}
SPL {X  -139.696, Y  +296.861, Z    +0.000, E1   +62.910, E3 +188743.469}
SPL {X  -137.330, Y  +293.030, Z    +0.000, E1   +62.290, E3 +188750.094}
SPL {X  -133.474, Y  +287.253, Z    +0.000, E1   +62.192, E3 +188755.833}
SPL {X  -124.928, Y  +276.081, Z    +0.000, E1   +64.269, E3 +188756.539}
SPL {X   -90.696, Y  +245.280, Z    +0.000, E1   +54.124, E3 +188877.257}
ENDSPLINE

SPLINE
SPL {X  -134.058, Y  +288.094, Z    +0.000, E1   +46.503, E3 +189004.771}
SPL {X  -153.979, Y  +327.577, Z    +0.000, E1   +33.452, E3 +189016.311}
SPL {X  -160.130, Y  +351.024, Z    +0.000, E1   +21.715, E3 +189020.741}
SPL {X  -162.127, Y  +365.491, Z    +0.000, E1   +12.692, E3 +189020.665}
SPL {X  -162.801, Y  +378.004, Z    +0.000, E1    +3.811, E3 +189021.081}
SPL {X  -162.820, Y  +382.997, Z    +0.000, E1    -0.389, E3 +189020.405}
SPL {X  -162.820, Y  +386.358, Z    +0.000, E1    -5.320, E3 +189020.140}
SPL {X  -162.820, Y  +390.608, Z    +0.000, E1   -12.198, E3 +189020.090}
SPL {X  -162.820, Y  +396.028, Z    +0.000, E1   -22.022, E3 +189019.958}
SPL {X  -162.820, Y  +402.037, Z    +0.000, E1   -32.247, E3 +189019.896}
SPL {X  -162.820, Y  +414.067, Z    +0.000, E1   -47.235, E3 +189021.322}
SPL {X  -162.820, Y  +424.566, Z    +0.000, E1   -59.255, E3 +189017.987}
SPL {X  -162.820, Y  +460.664, Z    +0.000, E1   -69.605, E3 +189026.284}
SPL {X  -162.820, Y  +481.040, Z    +0.000, E1   -67.047, E3 +189044.872}
SPL {X  -162.820, Y  +576.352, Z    +0.000, E1   -67.140, E3 +189112.391}
ENDSPLINE

SPLINE
SPL {X  -162.820, Y  +573.336, Z    +0.000, E1   -64.995, E3 +189126.143}
ENDSPLINE

SPLINE
SPL {X  -162.820, Y  +580.233, Z    +0.000, E1   -64.427, E3 +189137.321}
SPL {X  -162.820, Y  +590.756, Z    +0.000, E1   -64.410, E3 +189147.889}
SPL {X  -162.820, Y  +600.605, Z    +0.000, E1   -64.446, E3 +189157.462}
SPL {X  -162.820, Y  +611.699, Z    +0.000, E1   -64.369, E3 +189169.142}
SPL {X  -162.820, Y  +625.950, Z    +0.000, E1   -64.427, E3 +189182.982}
SPL {X  -162.820, Y  +639.401, Z    +0.000, E1   -64.540, E3 +189195.404}
SPL {X  -162.820, Y  +648.933, Z    +0.000, E1   -64.417, E3 +189205.823}
SPL {X  -162.820, Y  +658.800, Z    +0.000, E1   -64.418, E3 +189215.637}
SPL {X  -162.820, Y  +670.777, Z    +0.000, E1   -64.432, E3 +189227.550}
SPL {X  -162.296, Y  +686.556, Z    +0.000, E1   -64.388, E3 +189243.753}
SPL {X  -160.469, Y  +701.070, Z    +0.000, E1   -64.058, E3 +189260.656}
SPL {X  -157.811, Y  +713.575, Z    +0.000, E1   -63.758, E3 +189275.235}
SPL {X  -154.601, Y  +724.576, Z    +0.000, E1   -63.303, E3 +189289.357}
SPL {X  -151.802, Y  +732.376, Z    +0.000, E1   -62.761, E3 +189300.485}
SPL {X  -149.758, Y  +737.398, Z    +0.000, E1   -62.434, E3 +189307.505}
SPL {X  -146.903, Y  +743.713, Z    +0.000, E1   -62.188, E3 +189315.278}
SPL {X  -144.901, Y  +747.758, Z    +0.000, E1   -61.566, E3 +189322.741}
SPL {X  -141.375, Y  +754.268, Z    +0.000, E1   -61.208, E3 +189331.295}
SPL {X  -137.988, Y  +759.927, Z    +0.000, E1   -60.537, E3 +189340.093}
SPL {X  -134.516, Y  +765.238, Z    +0.000, E1   -60.629, E3 +189344.896}
SPL {X  -126.113, Y  +776.485, Z    +0.000, E1   -62.672, E3 +189346.457}
SPL {X   -94.739, Y  +805.919, Z    +0.000, E1   -54.063, E3 +189453.198}
ENDSPLINE

SPLINE
SPL {X  -130.051, Y  +771.465, Z    +0.000, E1   -46.832, E3 +189574.982}
SPL {X  -150.288, Y  +736.141, Z    +0.000, E1   -36.889, E3 +189594.838}
SPL {X  -159.122, Y  +708.003, Z    +0.000, E1   -24.018, E3 +189597.546}
SPL {X  -161.938, Y  +690.423, Z    +0.000, E1   -13.625, E3 +189598.757}
SPL {X  -162.746, Y  +678.392, Z    +0.000, E1    -5.513, E3 +189598.830}
SPL {X  -162.820, Y  +672.097, Z    +0.000, E1    -0.584, E3 +189598.534}
SPL {X  -162.820, Y  +670.674, Z    +0.000, E1    +0.808, E3 +189598.166}
SPL {X  -162.820, Y  +666.307, Z    +0.000, E1    +6.851, E3 +189597.949}
SPL {X  -162.820, Y  +660.761, Z    +0.000, E1   +16.102, E3 +189598.092}
SPL {X  -162.820, Y  +655.024, Z    +0.000, E1   +25.730, E3 +189598.253}
SPL {X  -162.820, Y  +646.498, Z    +0.000, E1   +39.738, E3 +189596.774}
SPL {X  -162.820, Y  +637.711, Z    +0.000, E1   +46.793, E3 +189601.266}
SPL {X  -162.820, Y  +613.264, Z    +0.000, E1   +68.325, E3 +189593.464}
SPL {X  -162.820, Y  +583.199, Z    +0.000, E1   +66.160, E3 +189616.955}
SPL {X  -162.820, Y  +480.401, Z    +0.000, E1   +65.660, E3 +189697.846}
ENDSPLINE

SPLINE
SPL {X  -162.820, Y  +490.253, Z    +0.000, E1   +62.754, E3 +189709.609}
SPL {X  -162.820, Y  +505.887, Z    +0.000, E1   +58.743, E3 +189719.299}
ENDSPLINE

SPLINE
SPL {X  -162.820, Y  +492.515, Z    +0.000, E1   +59.352, E3 +189731.984}
SPL {X  -162.820, Y  +476.196, Z    +0.000, E1   +60.204, E3 +189746.017}
SPL {X  -162.820, Y  +460.138, Z    +0.000, E1   +61.014, E3 +189759.200}
SPL {X  -162.820, Y  +442.137, Z    +0.000, E1   +61.946, E3 +189773.096}
SPL {X  -162.820, Y  +425.982, Z    +0.000, E1   +62.713, E3 +189785.123}
SPL {X  -162.820, Y  +413.005, Z    +0.000, E1   +63.234, E3 +189795.137}
SPL {X  -162.820, Y  +396.727, Z    +0.000, E1   +63.972, E3 +189806.489}
SPL {X  -162.820, Y  +382.966, Z    +0.000, E1   +64.511, E3 +189816.211}
SPL {X  -161.867, Y  +362.911, Z    +0.000, E1   +65.480, E3 +189828.285}
SPL {X  -158.833, Y  +344.688, Z    +0.000, E1   +65.800, E3 +189842.785}
SPL {X  -155.590, Y  +332.521, Z    +0.000, E1   +65.288, E3 +189857.719}
SPL {X  -151.631, Y  +321.184, Z    +0.000, E1   +64.776, E3 +189871.572}
SPL {X  -147.832, Y  +312.265, Z    +0.000, E1   +64.201, E3 +189883.382}
SPL {X  -145.264, Y  +306.955, Z    +0.000, E1   +63.555, E3 +189891.988}
SPL {X  -142.454, Y  +301.650, Z    +0.000, E1   +63.360, E3 +189897.991}
SPL {X  -139.696, Y  +296.861, Z    +0.000, E1   +62.910, E3 +189904.759}
SPL {X  -137.330, Y  +293.030, Z    +0.000, E1   +62.290, E3 +189911.384}
SPL {X  -134.245, Y  +288.366, Z    +0.000, E1   +62.031, E3 +189916.865}
SPL {X  -128.642, Y  +280.693, Z    +0.000, E1   +63.351, E3 +189917.859}
SPL {X   -90.696, Y  +245.280, Z    +0.000, E1   +54.124, E3 +190038.548}
ENDSPLINE

SPLINE
SPL {X  -134.058, Y  +288.094, Z    +0.000, E1   +46.503, E3 +190166.061}
SPL {X  -153.979, Y  +327.577, Z    +0.000, E1   +33.452, E3 +190177.601}
SPL {X  -160.130, Y  +351.024, Z    +0.000, E1   +21.715, E3 +190182.032}
SPL {X  -162.127, Y  +365.491, Z    +0.000, E1   +12.692, E3 +190181.955}
SPL {X  -162.801, Y  +378.004, Z    +0.000, E1    +3.811, E3 +190182.371}
SPL {X  -162.820, Y  +382.501, Z    +0.000, E1    +0.028, E3 +190181.790}
SPL {X  -162.820, Y  +385.123, Z    +0.000, E1    -3.284, E3 +190181.467}
SPL {X  -162.820, Y  +390.608, Z    +0.000, E1   -12.198, E3 +190181.381}
SPL {X  -162.820, Y  +396.028, Z    +0.000, E1   -22.022, E3 +190181.249}
SPL {X  -162.820, Y  +402.037, Z    +0.000, E1   -32.247, E3 +190181.186}
SPL {X  -162.820, Y  +411.189, Z    +0.000, E1   -44.140, E3 +190182.516}
SPL {X  -162.820, Y  +422.160, Z    +0.000, E1   -56.042, E3 +190180.988}
SPL {X  -162.820, Y  +475.891, Z    +0.000, E1   -67.666, E3 +190201.306}
SPL {X  -162.820, Y  +573.811, Z    +0.000, E1   -65.269, E3 +190285.905}
SPL {X  -162.820, Y  +580.233, Z    +0.000, E1   -64.427, E3 +190298.611}
SPL {X  -162.820, Y  +590.756, Z    +0.000, E1   -64.410, E3 +190309.179}
SPL {X  -162.820, Y  +600.605, Z    +0.000, E1   -64.446, E3 +190318.752}
SPL {X  -162.820, Y  +611.699, Z    +0.000, E1   -64.369, E3 +190330.432}
SPL {X  -162.820, Y  +622.825, Z    +0.000, E1   -64.446, E3 +190340.876}
SPL {X  -162.820, Y  +635.776, Z    +0.000, E1   -64.495, E3 +190353.566}
SPL {X  -162.820, Y  +648.933, Z    +0.000, E1   -64.417, E3 +190367.113}
SPL {X  -162.820, Y  +658.800, Z    +0.000, E1   -64.418, E3 +190376.927}
SPL {X  -162.820, Y  +670.777, Z    +0.000, E1   -64.432, E3 +190388.841}
SPL {X  -162.296, Y  +686.556, Z    +0.000, E1   -64.388, E3 +190405.044}
SPL {X  -160.469, Y  +701.070, Z    +0.000, E1   -64.058, E3 +190421.947}
SPL {X  -157.811, Y  +713.575, Z    +0.000, E1   -63.758, E3 +190436.526}
SPL {X  -154.601, Y  +724.576, Z    +0.000, E1   -63.303, E3 +190450.648}
SPL {X  -151.802, Y  +732.376, Z    +0.000, E1   -62.761, E3 +190461.775}
SPL {X  -149.758, Y  +737.398, Z    +0.000, E1   -62.434, E3 +190468.795}
SPL {X  -146.903, Y  +743.713, Z    +0.000, E1   -62.188, E3 +190476.568}
SPL {X  -144.901, Y  +747.758, Z    +0.000, E1   -61.566, E3 +190484.031}
SPL {X  -141.375, Y  +754.268, Z    +0.000, E1   -61.208, E3 +190492.585}
SPL {X  -137.988, Y  +759.927, Z    +0.000, E1   -60.537, E3 +190501.383}
SPL {X  -133.449, Y  +766.783, Z    +0.000, E1   -60.899, E3 +190506.431}
SPL {X   -94.739, Y  +805.919, Z    +0.000, E1   -54.063, E3 +190614.488}
ENDSPLINE

SPLINE
SPL {X  -120.571, Y  +782.921, Z    +0.000, E1   -48.746, E3 +190721.784}
SPL {X  -145.902, Y  +745.770, Z    +0.000, E1   -40.275, E3 +190752.932}
SPL {X  -159.122, Y  +708.003, Z    +0.000, E1   -24.018, E3 +190758.836}
SPL {X  -161.938, Y  +690.423, Z    +0.000, E1   -13.625, E3 +190760.047}
SPL {X  -162.638, Y  +681.194, Z    +0.000, E1    -7.430, E3 +190759.868}
SPL {X  -162.820, Y  +672.793, Z    +0.000, E1    -1.263, E3 +190759.926}
SPL {X  -162.820, Y  +670.674, Z    +0.000, E1    +0.808, E3 +190759.457}
SPL {X  -162.820, Y  +666.307, Z    +0.000, E1    +6.851, E3 +190759.239}
SPL {X  -162.820, Y  +660.761, Z    +0.000, E1   +16.102, E3 +190759.382}
SPL {X  -162.820, Y  +655.024, Z    +0.000, E1   +25.730, E3 +190759.543}
SPL {X  -162.820, Y  +646.498, Z    +0.000, E1   +39.738, E3 +190758.064}
SPL {X  -162.820, Y  +637.711, Z    +0.000, E1   +46.793, E3 +190762.557}
SPL {X  -162.820, Y  +598.602, Z    +0.000, E1   +67.541, E3 +190765.108}
SPL {X  -162.820, Y  +578.435, Z    +0.000, E1   +65.472, E3 +190783.207}
SPL {X  -162.820, Y  +475.450, Z    +0.000, E1   +67.130, E3 +190852.145}
ENDSPLINE

SPLINE
SPL {X  -162.820, Y  +483.223, Z    +0.000, E1   +64.312, E3 +190866.585}
SPL {X  -162.820, Y  +502.830, Z    +0.000, E1   +59.229, E3 +190881.505}
ENDSPLINE

SPLINE
SPL {X  -162.820, Y  +486.621, Z    +0.000, E1   +59.661, E3 +190898.425}
SPL {X  -162.820, Y  +472.771, Z    +0.000, E1   +60.369, E3 +190910.170}
SPL {X  -162.820, Y  +460.138, Z    +0.000, E1   +61.014, E3 +190920.490}
SPL {X  -162.820, Y  +448.741, Z    +0.000, E1   +61.510, E3 +190930.005}
SPL {X  -162.820, Y  +430.985, Z    +0.000, E1   +62.533, E3 +190942.438}
SPL {X  -162.820, Y  +413.005, Z    +0.000, E1   +63.234, E3 +190956.428}
SPL {X  -162.820, Y  +396.727, Z    +0.000, E1   +63.972, E3 +190967.779}
SPL {X  -162.820, Y  +382.966, Z    +0.000, E1   +64.511, E3 +190977.501}
SPL {X  -161.867, Y  +362.911, Z    +0.000, E1   +65.480, E3 +190989.575}
SPL {X  -159.475, Y  +347.667, Z    +0.000, E1   +65.889, E3 +191000.494}
SPL {X  -157.043, Y  +337.513, Z    +0.000, E1   +65.541, E3 +191012.572}
SPL {X  -153.776, Y  +326.991, Z    +0.000, E1   +65.023, E3 +191025.812}
SPL {X  -149.992, Y  +317.154, Z    +0.000, E1   +64.515, E3 +191038.276}
SPL {X  -146.026, Y  +308.480, Z    +0.000, E1   +63.813, E3 +191050.518}
SPL {X  -142.454, Y  +301.650, Z    +0.000, E1   +63.360, E3 +191059.282}
SPL {X  -139.696, Y  +296.861, Z    +0.000, E1   +62.910, E3 +191066.049}
SPL {X  -137.330, Y  +293.030, Z    +0.000, E1   +62.290, E3 +191072.674}
SPL {X  -134.245, Y  +288.366, Z    +0.000, E1   +62.031, E3 +191078.156}
SPL {X  -128.642, Y  +280.693, Z    +0.000, E1   +63.351, E3 +191079.149}
SPL {X   -90.696, Y  +245.280, Z    +0.000, E1   +54.124, E3 +191199.838}
ENDSPLINE

SPLINE
SPL {X  -134.058, Y  +288.094, Z    +0.000, E1   +46.503, E3 +191327.351}
SPL {X  -148.633, Y  +314.028, Z    +0.000, E1   +38.752, E3 +191336.240}
SPL {X  -156.325, Y  +334.971, Z    +0.000, E1   +30.037, E3 +191340.008}
SPL {X  -160.130, Y  +351.024, Z    +0.000, E1   +21.715, E3 +191343.322}
SPL {X  -162.127, Y  +365.491, Z    +0.000, E1   +12.692, E3 +191343.246}
SPL {X  -162.801, Y  +378.004, Z    +0.000, E1    +3.811, E3 +191343.662}
SPL {X  -162.820, Y  +382.501, Z    +0.000, E1    +0.028, E3 +191343.080}
SPL {X  -162.820, Y  +385.123, Z    +0.000, E1    -3.284, E3 +191342.757}
SPL {X  -162.820, Y  +390.608, Z    +0.000, E1   -12.198, E3 +191342.671}
SPL {X  -162.820, Y  +396.028, Z    +0.000, E1   -22.022, E3 +191342.539}
SPL {X  -162.820, Y  +402.037, Z    +0.000, E1   -32.247, E3 +191342.477}
SPL {X  -162.820, Y  +411.189, Z    +0.000, E1   -44.140, E3 +191343.806}
SPL {X  -162.820, Y  +422.160, Z    +0.000, E1   -56.042, E3 +191342.278}
SPL {X  -162.820, Y  +475.891, Z    +0.000, E1   -67.666, E3 +191362.597}
SPL {X  -162.820, Y  +573.811, Z    +0.000, E1   -65.269, E3 +191447.195}
SPL {X  -162.820, Y  +580.233, Z    +0.000, E1   -64.427, E3 +191459.902}
SPL {X  -162.820, Y  +590.756, Z    +0.000, E1   -64.410, E3 +191470.469}
SPL {X  -162.820, Y  +600.605, Z    +0.000, E1   -64.446, E3 +191480.043}
SPL {X  -162.820, Y  +611.699, Z    +0.000, E1   -64.369, E3 +191491.722}
SPL {X  -162.820, Y  +622.825, Z    +0.000, E1   -64.446, E3 +191502.167}
SPL {X  -162.820, Y  +635.776, Z    +0.000, E1   -64.495, E3 +191514.856}
SPL {X  -162.820, Y  +648.933, Z    +0.000, E1   -64.417, E3 +191528.403}
SPL {X  -162.820, Y  +658.800, Z    +0.000, E1   -64.418, E3 +191538.218}
SPL {X  -162.820, Y  +670.777, Z    +0.000, E1   -64.432, E3 +191550.131}
SPL {X  -162.296, Y  +686.556, Z    +0.000, E1   -64.388, E3 +191566.334}
SPL {X  -160.469, Y  +701.070, Z    +0.000, E1   -64.058, E3 +191583.237}
SPL {X  -157.811, Y  +713.575, Z    +0.000, E1   -63.758, E3 +191597.816}
SPL {X  -155.696, Y  +721.135, Z    +0.000, E1   -63.387, E3 +191607.749}
SPL {X  -153.915, Y  +726.609, Z    +0.000, E1   -63.196, E3 +191614.524}
SPL {X  -151.802, Y  +732.376, Z    +0.000, E1   -62.761, E3 +191623.065}
SPL {X  -149.758, Y  +737.398, Z    +0.000, E1   -62.434, E3 +191630.086}
SPL {X  -146.903, Y  +743.713, Z    +0.000, E1   -62.188, E3 +191637.858}
SPL {X  -143.515, Y  +750.401, Z    +0.000, E1   -61.484, E3 +191648.543}
SPL {X  -140.303, Y  +756.116, Z    +0.000, E1   -60.974, E3 +191656.740}
SPL {X  -137.988, Y  +759.927, Z    +0.000, E1   -60.537, E3 +191662.674}
SPL {X  -134.516, Y  +765.238, Z    +0.000, E1   -60.629, E3 +191667.477}
SPL {X  -126.113, Y  +776.485, Z    +0.000, E1   -62.672, E3 +191669.038}
SPL {X   -95.040, Y  +805.704, Z    +0.000, E1   -55.103, E3 +191759.997}
ENDSPLINE

SPLINE
SPL {X   -95.634, Y  +805.274, Z    +0.000, E1   -52.767, E3 +191799.156}
SPL {X  -130.051, Y  +771.465, Z    +0.000, E1   -46.832, E3 +191897.562}
SPL {X  -154.243, Y  +725.647, Z    +0.000, E1   -32.659, E3 +191919.125}
SPL {X  -160.324, Y  +701.901, Z    +0.000, E1   -20.534, E3 +191919.947}
SPL {X  -161.938, Y  +690.423, Z    +0.000, E1   -13.625, E3 +191921.338}
SPL {X  -162.746, Y  +678.392, Z    +0.000, E1    -5.513, E3 +191921.410}
SPL {X  -162.820, Y  +671.700, Z    +0.000, E1    -0.272, E3 +191920.976}
SPL {X  -162.820, Y  +668.888, Z    +0.000, E1    +3.063, E3 +191920.673}
SPL {X  -162.820, Y  +664.763, Z    +0.000, E1    +9.526, E3 +191920.333}
SPL {X  -162.820, Y  +660.761, Z    +0.000, E1   +16.102, E3 +191920.672}
SPL {X  -162.820, Y  +655.024, Z    +0.000, E1   +25.730, E3 +191920.833}
SPL {X  -162.820, Y  +646.498, Z    +0.000, E1   +39.738, E3 +191919.354}
SPL {X  -162.820, Y  +637.711, Z    +0.000, E1   +46.793, E3 +191923.847}
SPL {X  -162.820, Y  +598.602, Z    +0.000, E1   +67.541, E3 +191926.398}
SPL {X  -162.820, Y  +578.435, Z    +0.000, E1   +65.472, E3 +191944.498}
SPL {X  -162.820, Y  +475.450, Z    +0.000, E1   +67.130, E3 +192013.435}
ENDSPLINE

SPLINE
SPL {X  -162.820, Y  +483.223, Z    +0.000, E1   +64.312, E3 +192027.875}
SPL {X  -162.820, Y  +502.830, Z    +0.000, E1   +59.229, E3 +192042.796}
ENDSPLINE

SPLINE
SPL {X  -162.820, Y  +486.621, Z    +0.000, E1   +59.661, E3 +192059.715}
SPL {X  -162.820, Y  +472.771, Z    +0.000, E1   +60.369, E3 +192071.461}
SPL {X  -162.820, Y  +460.138, Z    +0.000, E1   +61.014, E3 +192081.780}
SPL {X  -162.820, Y  +448.741, Z    +0.000, E1   +61.510, E3 +192091.295}
SPL {X  -162.820, Y  +430.985, Z    +0.000, E1   +62.533, E3 +192103.728}
SPL {X  -162.820, Y  +413.005, Z    +0.000, E1   +63.234, E3 +192117.718}
SPL {X  -162.820, Y  +396.727, Z    +0.000, E1   +63.972, E3 +192129.069}
SPL {X  -162.756, Y  +375.937, Z    +0.000, E1   +64.914, E3 +192142.679}
SPL {X  -161.353, Y  +358.691, Z    +0.000, E1   +65.588, E3 +192153.903}
SPL {X  -158.833, Y  +344.688, Z    +0.000, E1   +65.800, E3 +192165.366}
SPL {X  -156.326, Y  +334.977, Z    +0.000, E1   +65.428, E3 +192176.839}
SPL {X  -153.776, Y  +326.991, Z    +0.000, E1   +65.023, E3 +192187.102}
SPL {X  -149.992, Y  +317.154, Z    +0.000, E1   +64.515, E3 +192199.566}
SPL {X  -146.026, Y  +308.480, Z    +0.000, E1   +63.813, E3 +192211.808}
SPL {X  -142.454, Y  +301.650, Z    +0.000, E1   +63.360, E3 +192220.572}
SPL {X  -139.696, Y  +296.861, Z    +0.000, E1   +62.910, E3 +192227.340}
SPL {X  -137.330, Y  +293.030, Z    +0.000, E1   +62.290, E3 +192233.965}
SPL {X  -134.245, Y  +288.366, Z    +0.000, E1   +62.031, E3 +192239.446}
SPL {X  -128.642, Y  +280.693, Z    +0.000, E1   +63.351, E3 +192240.439}
SPL {X   -90.696, Y  +245.280, Z    +0.000, E1   +54.124, E3 +192361.128}
ENDSPLINE

SPLINE
SPL {X  -134.058, Y  +288.094, Z    +0.000, E1   +46.503, E3 +192488.642}
SPL {X  -153.979, Y  +327.577, Z    +0.000, E1   +33.452, E3 +192500.182}
SPL {X  -160.130, Y  +351.024, Z    +0.000, E1   +21.715, E3 +192504.612}
SPL {X  -162.127, Y  +365.491, Z    +0.000, E1   +12.692, E3 +192504.536}
SPL {X  -162.801, Y  +378.004, Z    +0.000, E1    +3.811, E3 +192504.952}
SPL {X  -162.820, Y  +382.501, Z    +0.000, E1    +0.028, E3 +192504.371}
SPL {X  -162.820, Y  +385.123, Z    +0.000, E1    -3.284, E3 +192504.048}
SPL {X  -162.820, Y  +390.608, Z    +0.000, E1   -12.198, E3 +192503.961}
SPL {X  -162.820, Y  +396.028, Z    +0.000, E1   -22.022, E3 +192503.829}
SPL {X  -162.820, Y  +402.037, Z    +0.000, E1   -32.247, E3 +192503.767}
SPL {X  -162.820, Y  +411.189, Z    +0.000, E1   -44.140, E3 +192505.097}
SPL {X  -162.820, Y  +422.160, Z    +0.000, E1   -56.042, E3 +192503.568}
SPL {X  -162.820, Y  +475.891, Z    +0.000, E1   -67.666, E3 +192523.887}
SPL {X  -162.820, Y  +573.811, Z    +0.000, E1   -65.269, E3 +192608.485}
SPL {X  -162.820, Y  +580.233, Z    +0.000, E1   -64.427, E3 +192621.192}
SPL {X  -162.820, Y  +590.756, Z    +0.000, E1   -64.410, E3 +192631.760}
SPL {X  -162.820, Y  +600.605, Z    +0.000, E1   -64.446, E3 +192641.333}
SPL {X  -162.820, Y  +611.699, Z    +0.000, E1   -64.369, E3 +192653.013}
SPL {X  -162.820, Y  +622.825, Z    +0.000, E1   -64.446, E3 +192663.457}
SPL {X  -162.820, Y  +635.776, Z    +0.000, E1   -64.495, E3 +192676.147}
SPL {X  -162.820, Y  +648.933, Z    +0.000, E1   -64.417, E3 +192689.694}
SPL {X  -162.820, Y  +658.800, Z    +0.000, E1   -64.418, E3 +192699.508}
SPL {X  -162.820, Y  +670.777, Z    +0.000, E1   -64.432, E3 +192711.421}
SPL {X  -162.296, Y  +686.556, Z    +0.000, E1   -64.388, E3 +192727.624}
SPL {X  -160.469, Y  +701.070, Z    +0.000, E1   -64.058, E3 +192744.527}
SPL {X  -157.811, Y  +713.575, Z    +0.000, E1   -63.758, E3 +192759.106}
SPL {X  -154.601, Y  +724.576, Z    +0.000, E1   -63.303, E3 +192773.228}
SPL {X  -151.802, Y  +732.376, Z    +0.000, E1   -62.761, E3 +192784.356}
SPL {X  -149.758, Y  +737.398, Z    +0.000, E1   -62.434, E3 +192791.376}
SPL {X  -146.903, Y  +743.713, Z    +0.000, E1   -62.188, E3 +192799.149}
SPL {X  -143.515, Y  +750.401, Z    +0.000, E1   -61.484, E3 +192809.833}
SPL {X  -138.985, Y  +758.314, Z    +0.000, E1   -60.770, E3 +192821.392}
SPL {X  -133.449, Y  +766.783, Z    +0.000, E1   -60.899, E3 +192829.012}
SPL {X   -94.739, Y  +805.919, Z    +0.000, E1   -54.063, E3 +192937.069}
ENDSPLINE

SPLINE
SPL {X  -130.051, Y  +771.465, Z    +0.000, E1   -46.832, E3 +193058.853}
SPL {X  -154.243, Y  +725.647, Z    +0.000, E1   -32.659, E3 +193080.415}
SPL {X  -160.324, Y  +701.901, Z    +0.000, E1   -20.534, E3 +193081.238}
SPL {X  -161.938, Y  +690.423, Z    +0.000, E1   -13.625, E3 +193082.628}
SPL {X  -162.638, Y  +681.194, Z    +0.000, E1    -7.430, E3 +193082.449}
SPL {X  -162.820, Y  +672.793, Z    +0.000, E1    -1.263, E3 +193082.507}
SPL {X  -162.820, Y  +670.674, Z    +0.000, E1    +0.808, E3 +193082.037}
SPL {X  -162.820, Y  +666.307, Z    +0.000, E1    +6.851, E3 +193081.820}
SPL {X  -162.820, Y  +660.761, Z    +0.000, E1   +16.102, E3 +193081.963}
SPL {X  -162.820, Y  +655.024, Z    +0.000, E1   +25.730, E3 +193082.124}
SPL {X  -162.820, Y  +646.498, Z    +0.000, E1   +39.738, E3 +193080.645}
SPL {X  -162.820, Y  +637.711, Z    +0.000, E1   +46.793, E3 +193085.137}
SPL {X  -162.820, Y  +598.602, Z    +0.000, E1   +67.541, E3 +193087.688}
SPL {X  -162.820, Y  +578.435, Z    +0.000, E1   +65.472, E3 +193105.788}
SPL {X  -162.820, Y  +480.401, Z    +0.000, E1   +65.660, E3 +193181.717}
ENDSPLINE

SPLINE
SPL {X  -162.820, Y  +490.253, Z    +0.000, E1   +62.754, E3 +193193.480}
SPL {X  -162.820, Y  +503.236, Z    +0.000, E1   +58.858, E3 +193205.833}
ENDSPLINE

SPLINE
SPL {X  -162.820, Y  +486.621, Z    +0.000, E1   +59.661, E3 +193221.006}
SPL {X  -162.820, Y  +472.771, Z    +0.000, E1   +60.369, E3 +193232.751}
SPL {X  -162.820, Y  +460.138, Z    +0.000, E1   +61.014, E3 +193243.071}
SPL {X  -162.820, Y  +448.741, Z    +0.000, E1   +61.510, E3 +193252.585}
SPL {X  -162.820, Y  +430.985, Z    +0.000, E1   +62.533, E3 +193265.018}
SPL {X  -162.820, Y  +413.005, Z    +0.000, E1   +63.234, E3 +193279.008}
SPL {X  -162.820, Y  +396.727, Z    +0.000, E1   +63.972, E3 +193290.360}
SPL {X  -162.756, Y  +375.937, Z    +0.000, E1   +64.914, E3 +193303.969}
SPL {X  -161.353, Y  +358.691, Z    +0.000, E1   +65.588, E3 +193315.194}
SPL {X  -159.475, Y  +347.667, Z    +0.000, E1   +65.889, E3 +193323.074}
SPL {X  -157.043, Y  +337.513, Z    +0.000, E1   +65.541, E3 +193335.152}
SPL {X  -154.736, Y  +329.832, Z    +0.000, E1   +65.034, E3 +193345.598}
SPL {X  -151.631, Y  +321.184, Z    +0.000, E1   +64.776, E3 +193355.443}
SPL {X  -147.832, Y  +312.265, Z    +0.000, E1   +64.201, E3 +193367.252}
SPL {X  -145.264, Y  +306.955, Z    +0.000, E1   +63.555, E3 +193375.858}
SPL {X  -142.454, Y  +301.650, Z    +0.000, E1   +63.360, E3 +193381.862}
SPL {X  -139.696, Y  +296.861, Z    +0.000, E1   +62.910, E3 +193388.630}
SPL {X  -137.330, Y  +293.030, Z    +0.000, E1   +62.290, E3 +193395.255}
SPL {X  -134.245, Y  +288.366, Z    +0.000, E1   +62.031, E3 +193400.736}
SPL {X  -128.642, Y  +280.693, Z    +0.000, E1   +63.351, E3 +193401.730}
SPL {X   -90.696, Y  +245.280, Z    +0.000, E1   +54.124, E3 +193522.418}
ENDSPLINE

SPLINE
SPL {X  -134.058, Y  +288.094, Z    +0.000, E1   +46.503, E3 +193649.932}
SPL {X  -153.979, Y  +327.577, Z    +0.000, E1   +33.452, E3 +193661.472}
SPL {X  -160.130, Y  +351.024, Z    +0.000, E1   +21.715, E3 +193665.903}
SPL {X  -162.127, Y  +365.491, Z    +0.000, E1   +12.692, E3 +193665.826}
SPL {X  -162.745, Y  +375.564, Z    +0.000, E1    +5.577, E3 +193666.437}
SPL {X  -162.820, Y  +382.222, Z    +0.000, E1    +0.380, E3 +193665.709}
SPL {X  -162.820, Y  +384.010, Z    +0.000, E1    -1.878, E3 +193665.372}
SPL {X  -162.820, Y  +387.631, Z    +0.000, E1    -7.169, E3 +193665.325}
SPL {X  -162.820, Y  +394.064, Z    +0.000, E1   -18.298, E3 +193665.136}
SPL {X  -162.820, Y  +402.037, Z    +0.000, E1   -32.247, E3 +193665.057}
SPL {X  -162.820, Y  +411.189, Z    +0.000, E1   -44.140, E3 +193666.387}
SPL {X  -162.820, Y  +422.160, Z    +0.000, E1   -56.042, E3 +193664.859}
SPL {X  -162.820, Y  +475.891, Z    +0.000, E1   -67.666, E3 +193685.177}
SPL {X  -162.820, Y  +573.811, Z    +0.000, E1   -65.269, E3 +193769.776}
SPL {X  -162.820, Y  +580.233, Z    +0.000, E1   -64.427, E3 +193782.482}
SPL {X  -162.820, Y  +590.756, Z    +0.000, E1   -64.410, E3 +193793.050}
SPL {X  -162.820, Y  +600.605, Z    +0.000, E1   -64.446, E3 +193802.623}
SPL {X  -162.820, Y  +611.699, Z    +0.000, E1   -64.369, E3 +193814.303}
SPL {X  -162.820, Y  +622.825, Z    +0.000, E1   -64.446, E3 +193824.747}
SPL {X  -162.820, Y  +635.776, Z    +0.000, E1   -64.495, E3 +193837.437}
SPL {X  -162.820, Y  +648.933, Z    +0.000, E1   -64.417, E3 +193850.984}
SPL {X  -162.820, Y  +658.800, Z    +0.000, E1   -64.418, E3 +193860.798}
SPL {X  -162.820, Y  +670.777, Z    +0.000, E1   -64.432, E3 +193872.712}
SPL {X  -162.296, Y  +686.556, Z    +0.000, E1   -64.388, E3 +193888.915}
SPL {X  -160.469, Y  +701.070, Z    +0.000, E1   -64.058, E3 +193905.818}
SPL {X  -157.811, Y  +713.575, Z    +0.000, E1   -63.758, E3 +193920.397}
SPL {X  -155.696, Y  +721.135, Z    +0.000, E1   -63.387, E3 +193930.330}
SPL {X  -153.915, Y  +726.609, Z    +0.000, E1   -63.196, E3 +193937.105}
SPL {X  -151.802, Y  +732.376, Z    +0.000, E1   -62.761, E3 +193945.646}
SPL {X  -149.758, Y  +737.398, Z    +0.000, E1   -62.434, E3 +193952.666}
SPL {X  -146.903, Y  +743.713, Z    +0.000, E1   -62.188, E3 +193960.439}
SPL {X  -144.901, Y  +747.758, Z    +0.000, E1   -61.566, E3 +193967.902}
SPL {X  -141.375, Y  +754.268, Z    +0.000, E1   -61.208, E3 +193976.456}
SPL {X  -137.124, Y  +761.291, Z    +0.000, E1   -60.398, E3 +193987.368}
SPL {X  -130.896, Y  +770.333, Z    +0.000, E1   -61.755, E3 +193990.042}
SPL {X   -94.739, Y  +805.919, Z    +0.000, E1   -54.063, E3 +194098.359}
ENDSPLINE

SPLINE
SPL {X  -130.051, Y  +771.465, Z    +0.000, E1   -46.832, E3 +194220.143}
SPL {X  -150.288, Y  +736.141, Z    +0.000, E1   -36.889, E3 +194239.999}
SPL {X  -159.122, Y  +708.003, Z    +0.000, E1   -24.018, E3 +194242.707}
SPL {X  -161.938, Y  +690.423, Z    +0.000, E1   -13.625, E3 +194243.918}
SPL {X  -162.746, Y  +678.392, Z    +0.000, E1    -5.513, E3 +194243.991}
SPL {X  -162.820, Y  +671.700, Z    +0.000, E1    -0.272, E3 +194243.557}
SPL {X  -162.820, Y  +668.888, Z    +0.000, E1    +3.063, E3 +194243.254}
SPL {X  -162.820, Y  +664.763, Z    +0.000, E1    +9.526, E3 +194242.913}
SPL {X  -162.820, Y  +660.761, Z    +0.000, E1   +16.102, E3 +194243.253}
SPL {X  -162.820, Y  +655.024, Z    +0.000, E1   +25.730, E3 +194243.414}
SPL {X  -162.820, Y  +646.498, Z    +0.000, E1   +39.738, E3 +194241.935}
SPL {X  -162.820, Y  +637.711, Z    +0.000, E1   +46.793, E3 +194246.428}
SPL {X  -162.820, Y  +613.264, Z    +0.000, E1   +68.325, E3 +194238.626}
SPL {X  -162.820, Y  +583.199, Z    +0.000, E1   +66.160, E3 +194262.116}
SPL {X  -162.820, Y  +480.401, Z    +0.000, E1   +65.660, E3 +194343.008}
ENDSPLINE

SPLINE
SPL {X  -162.820, Y  +490.253, Z    +0.000, E1   +62.754, E3 +194354.770}
SPL {X  -162.820, Y  +503.236, Z    +0.000, E1   +58.858, E3 +194367.124}
ENDSPLINE

SPLINE
SPL {X  -162.820, Y  +486.621, Z    +0.000, E1   +59.661, E3 +194382.296}
SPL {X  -162.820, Y  +472.771, Z    +0.000, E1   +60.369, E3 +194394.041}
SPL {X  -162.820, Y  +460.138, Z    +0.000, E1   +61.014, E3 +194404.361}
SPL {X  -162.820, Y  +448.741, Z    +0.000, E1   +61.510, E3 +194413.876}
SPL {X  -162.820, Y  +430.985, Z    +0.000, E1   +62.533, E3 +194426.309}
SPL {X  -162.820, Y  +413.005, Z    +0.000, E1   +63.234, E3 +194440.299}
SPL {X  -162.820, Y  +396.727, Z    +0.000, E1   +63.972, E3 +194451.650}
SPL {X  -162.756, Y  +375.937, Z    +0.000, E1   +64.914, E3 +194465.259}
SPL {X  -161.353, Y  +358.691, Z    +0.000, E1   +65.588, E3 +194476.484}
SPL {X  -159.475, Y  +347.667, Z    +0.000, E1   +65.889, E3 +194484.365}
SPL {X  -157.043, Y  +337.513, Z    +0.000, E1   +65.541, E3 +194496.442}
SPL {X  -153.776, Y  +326.991, Z    +0.000, E1   +65.023, E3 +194509.683}
SPL {X  -149.992, Y  +317.154, Z    +0.000, E1   +64.515, E3 +194522.147}
SPL {X  -146.026, Y  +308.480, Z    +0.000, E1   +63.813, E3 +194534.389}
SPL {X  -142.454, Y  +301.650, Z    +0.000, E1   +63.360, E3 +194543.153}
SPL {X  -139.696, Y  +296.861, Z    +0.000, E1   +62.910, E3 +194549.920}
SPL {X  -137.330, Y  +293.030, Z    +0.000, E1   +62.290, E3 +194556.545}
SPL {X  -134.245, Y  +288.366, Z    +0.000, E1   +62.031, E3 +194562.027}
SPL {X  -128.642, Y  +280.693, Z    +0.000, E1   +63.351, E3 +194563.020}
SPL {X   -90.696, Y  +245.280, Z    +0.000, E1   +54.124, E3 +194683.709}
ENDSPLINE

SPLINE
SPL {X  -134.058, Y  +288.094, Z    +0.000, E1   +46.503, E3 +194811.222}
SPL {X  -148.633, Y  +314.028, Z    +0.000, E1   +38.752, E3 +194820.111}
SPL {X  -156.325, Y  +334.971, Z    +0.000, E1   +30.037, E3 +194823.879}
SPL {X  -160.130, Y  +351.024, Z    +0.000, E1   +21.715, E3 +194827.193}
SPL {X  -162.127, Y  +365.491, Z    +0.000, E1   +12.692, E3 +194827.117}
SPL {X  -162.801, Y  +378.004, Z    +0.000, E1    +3.811, E3 +194827.533}
SPL {X  -162.820, Y  +382.997, Z    +0.000, E1    -0.389, E3 +194826.856}
SPL {X  -162.820, Y  +386.358, Z    +0.000, E1    -5.320, E3 +194826.591}
SPL {X  -162.820, Y  +390.608, Z    +0.000, E1   -12.198, E3 +194826.542}
SPL {X  -162.820, Y  +396.028, Z    +0.000, E1   -22.022, E3 +194826.410}
SPL {X  -162.820, Y  +402.037, Z    +0.000, E1   -32.247, E3 +194826.348}
SPL {X  -162.820, Y  +411.189, Z    +0.000, E1   -44.140, E3 +194827.677}
SPL {X  -162.820, Y  +422.160, Z    +0.000, E1   -56.042, E3 +194826.149}
SPL {X  -162.820, Y  +475.891, Z    +0.000, E1   -67.666, E3 +194846.468}
SPL {X  -162.820, Y  +576.352, Z    +0.000, E1   -67.140, E3 +194918.842}
ENDSPLINE

SPLINE
SPL {X  -162.820, Y  +573.336, Z    +0.000, E1   -64.995, E3 +194932.594}
ENDSPLINE

SPLINE
SPL {X  -162.820, Y  +580.233, Z    +0.000, E1   -64.427, E3 +194943.773}
SPL {X  -162.820, Y  +590.756, Z    +0.000, E1   -64.410, E3 +194954.340}
SPL {X  -162.820, Y  +600.605, Z    +0.000, E1   -64.446, E3 +194963.914}
SPL {X  -162.820, Y  +611.699, Z    +0.000, E1   -64.369, E3 +194975.593}
SPL {X  -162.820, Y  +625.950, Z    +0.000, E1   -64.427, E3 +194989.433}
SPL {X  -162.820, Y  +639.401, Z    +0.000, E1   -64.540, E3 +195001.856}
SPL {X  -162.820, Y  +648.933, Z    +0.000, E1   -64.417, E3 +195012.274}
SPL {X  -162.820, Y  +658.800, Z    +0.000, E1   -64.418, E3 +195022.089}
SPL {X  -162.820, Y  +670.777, Z    +0.000, E1   -64.432, E3 +195034.002}
SPL {X  -162.296, Y  +686.556, Z    +0.000, E1   -64.388, E3 +195050.205}
SPL {X  -161.171, Y  +696.611, Z    +0.000, E1   -64.029, E3 +195062.670}
SPL {X  -159.311, Y  +707.123, Z    +0.000, E1   -64.022, E3 +195073.364}
SPL {X  -156.625, Y  +717.984, Z    +0.000, E1   -63.524, E3 +195087.719}
SPL {X  -153.915, Y  +726.609, Z    +0.000, E1   -63.196, E3 +195098.395}
SPL {X  -151.802, Y  +732.376, Z    +0.000, E1   -62.761, E3 +195106.936}
SPL {X  -149.758, Y  +737.398, Z    +0.000, E1   -62.434, E3 +195113.957}
SPL {X  -146.903, Y  +743.713, Z    +0.000, E1   -62.188, E3 +195121.729}
SPL {X  -143.515, Y  +750.401, Z    +0.000, E1   -61.484, E3 +195132.414}
SPL {X  -140.303, Y  +756.116, Z    +0.000, E1   -60.974, E3 +195140.611}
SPL {X  -137.124, Y  +761.291, Z    +0.000, E1   -60.398, E3 +195148.658}
SPL {X  -130.896, Y  +770.333, Z    +0.000, E1   -61.755, E3 +195151.332}
SPL {X   -94.739, Y  +805.919, Z    +0.000, E1   -54.063, E3 +195259.649}
ENDSPLINE

SPLINE
SPL {X  -130.051, Y  +771.465, Z    +0.000, E1   -46.832, E3 +195381.433}
SPL {X  -154.243, Y  +725.647, Z    +0.000, E1   -32.659, E3 +195402.995}
SPL {X  -161.394, Y  +695.005, Z    +0.000, E1   -16.571, E3 +195404.700}
SPL {X  -162.746, Y  +678.392, Z    +0.000, E1    -5.513, E3 +195405.281}
SPL {X  -162.820, Y  +671.700, Z    +0.000, E1    -0.272, E3 +195404.847}
SPL {X  -162.820, Y  +669.993, Z    +0.000, E1    +1.755, E3 +195404.514}
SPL {X  -162.820, Y  +666.307, Z    +0.000, E1    +6.851, E3 +195404.400}
SPL {X  -162.820, Y  +660.761, Z    +0.000, E1   +16.102, E3 +195404.543}
SPL {X  -162.820, Y  +655.024, Z    +0.000, E1   +25.730, E3 +195404.704}
SPL {X  -162.820, Y  +646.498, Z    +0.000, E1   +39.738, E3 +195403.225}
SPL {X  -162.820, Y  +637.711, Z    +0.000, E1   +46.793, E3 +195407.718}
SPL {X  -162.820, Y  +613.264, Z    +0.000, E1   +68.325, E3 +195399.916}
SPL {X  -162.820, Y  +583.199, Z    +0.000, E1   +66.160, E3 +195423.407}
SPL {X  -162.820, Y  +480.401, Z    +0.000, E1   +65.660, E3 +195504.298}
ENDSPLINE

SPLINE
SPL {X  -162.820, Y  +490.253, Z    +0.000, E1   +62.754, E3 +195516.060}
SPL {X  -162.820, Y  +505.887, Z    +0.000, E1   +58.743, E3 +195525.751}
ENDSPLINE

SPLINE
SPL {X  -162.820, Y  +492.515, Z    +0.000, E1   +59.352, E3 +195538.436}
SPL {X  -162.820, Y  +476.196, Z    +0.000, E1   +60.204, E3 +195552.469}
SPL {X  -162.820, Y  +460.138, Z    +0.000, E1   +61.014, E3 +195565.651}
SPL {X  -162.820, Y  +448.741, Z    +0.000, E1   +61.510, E3 +195575.166}
SPL {X  -162.820, Y  +430.985, Z    +0.000, E1   +62.533, E3 +195587.599}
SPL {X  -162.820, Y  +413.005, Z    +0.000, E1   +63.234, E3 +195601.589}
SPL {X  -162.820, Y  +396.727, Z    +0.000, E1   +63.972, E3 +195612.940}
SPL {X  -162.756, Y  +375.937, Z    +0.000, E1   +64.914, E3 +195626.550}
SPL {X  -161.353, Y  +358.691, Z    +0.000, E1   +65.588, E3 +195637.774}
SPL {X  -158.833, Y  +344.688, Z    +0.000, E1   +65.800, E3 +195649.237}
SPL {X  -156.326, Y  +334.977, Z    +0.000, E1   +65.428, E3 +195660.710}
SPL {X  -153.776, Y  +326.991, Z    +0.000, E1   +65.023, E3 +195670.973}
SPL {X  -150.991, Y  +319.573, Z    +0.000, E1   +64.614, E3 +195680.427}
SPL {X  -147.832, Y  +312.265, Z    +0.000, E1   +64.201, E3 +195689.833}
SPL {X  -145.264, Y  +306.955, Z    +0.000, E1   +63.555, E3 +195698.439}
SPL {X  -142.454, Y  +301.650, Z    +0.000, E1   +63.360, E3 +195704.443}
SPL {X  -139.696, Y  +296.861, Z    +0.000, E1   +62.910, E3 +195711.211}
SPL {X  -137.330, Y  +293.030, Z    +0.000, E1   +62.290, E3 +195717.835}
SPL {X  -134.245, Y  +288.366, Z    +0.000, E1   +62.031, E3 +195723.317}
SPL {X  -128.642, Y  +280.693, Z    +0.000, E1   +63.351, E3 +195724.310}
SPL {X   -90.696, Y  +245.280, Z    +0.000, E1   +54.124, E3 +195844.999}
ENDSPLINE

SPLINE
SPL {X  -134.058, Y  +288.094, Z    +0.000, E1   +46.503, E3 +195972.513}
SPL {X  -153.979, Y  +327.577, Z    +0.000, E1   +33.452, E3 +195984.053}
SPL {X  -160.130, Y  +351.024, Z    +0.000, E1   +21.715, E3 +195988.483}
SPL {X  -162.127, Y  +365.491, Z    +0.000, E1   +12.692, E3 +195988.407}
SPL {X  -162.801, Y  +378.004, Z    +0.000, E1    +3.811, E3 +195988.823}
SPL {X  -162.820, Y  +382.501, Z    +0.000, E1    +0.028, E3 +195988.241}
SPL {X  -162.820, Y  +384.010, Z    +0.000, E1    -1.878, E3 +195987.952}
SPL {X  -162.820, Y  +387.631, Z    +0.000, E1    -7.169, E3 +195987.906}
SPL {X  -162.820, Y  +394.064, Z    +0.000, E1   -18.298, E3 +195987.716}
SPL {X  -162.820, Y  +402.037, Z    +0.000, E1   -32.247, E3 +195987.638}
SPL {X  -162.820, Y  +411.189, Z    +0.000, E1   -44.140, E3 +195988.968}
SPL {X  -162.820, Y  +422.160, Z    +0.000, E1   -56.042, E3 +195987.439}
SPL {X  -162.820, Y  +475.891, Z    +0.000, E1   -67.666, E3 +196007.758}
SPL {X  -162.820, Y  +573.811, Z    +0.000, E1   -65.269, E3 +196092.356}
SPL {X  -162.820, Y  +580.233, Z    +0.000, E1   -64.427, E3 +196105.063}
SPL {X  -162.820, Y  +590.756, Z    +0.000, E1   -64.410, E3 +196115.631}
SPL {X  -162.820, Y  +600.605, Z    +0.000, E1   -64.446, E3 +196125.204}
SPL {X  -162.820, Y  +611.699, Z    +0.000, E1   -64.369, E3 +196136.884}
SPL {X  -162.820, Y  +625.950, Z    +0.000, E1   -64.427, E3 +196150.724}
SPL {X  -162.820, Y  +639.401, Z    +0.000, E1   -64.540, E3 +196163.146}
SPL {X  -162.820, Y  +648.933, Z    +0.000, E1   -64.417, E3 +196173.565}
SPL {X  -162.820, Y  +658.800, Z    +0.000, E1   -64.418, E3 +196183.379}
SPL {X  -162.820, Y  +670.777, Z    +0.000, E1   -64.432, E3 +196195.292}
SPL {X  -162.613, Y  +681.710, Z    +0.000, E1   -64.310, E3 +196207.056}
SPL {X  -161.587, Y  +693.503, Z    +0.000, E1   -64.259, E3 +196219.410}
SPL {X  -159.311, Y  +707.123, Z    +0.000, E1   -64.022, E3 +196234.654}
SPL {X  -156.625, Y  +717.984, Z    +0.000, E1   -63.524, E3 +196249.009}
SPL {X  -153.915, Y  +726.609, Z    +0.000, E1   -63.196, E3 +196259.685}
SPL {X  -151.802, Y  +732.376, Z    +0.000, E1   -62.761, E3 +196268.227}
SPL {X  -149.758, Y  +737.398, Z    +0.000, E1   -62.434, E3 +196275.247}
SPL {X  -146.903, Y  +743.713, Z    +0.000, E1   -62.188, E3 +196283.020}
SPL {X  -143.515, Y  +750.401, Z    +0.000, E1   -61.484, E3 +196293.704}
SPL {X  -140.303, Y  +756.116, Z    +0.000, E1   -60.974, E3 +196301.902}
SPL {X  -137.988, Y  +759.927, Z    +0.000, E1   -60.537, E3 +196307.835}
SPL {X  -134.516, Y  +765.238, Z    +0.000, E1   -60.629, E3 +196312.638}
SPL {X  -126.113, Y  +776.485, Z    +0.000, E1   -62.672, E3 +196314.199}
SPL {X   -94.739, Y  +805.919, Z    +0.000, E1   -54.063, E3 +196420.940}
ENDSPLINE

SPLINE
SPL {X  -130.051, Y  +771.465, Z    +0.000, E1   -46.832, E3 +196542.724}
SPL {X  -154.243, Y  +725.647, Z    +0.000, E1   -32.659, E3 +196564.286}
SPL {X  -160.324, Y  +701.901, Z    +0.000, E1   -20.534, E3 +196565.109}
SPL {X  -161.938, Y  +690.423, Z    +0.000, E1   -13.625, E3 +196566.499}
SPL {X  -162.638, Y  +681.194, Z    +0.000, E1    -7.430, E3 +196566.320}
SPL {X  -162.805, Y  +675.686, Z    +0.000, E1    -3.400, E3 +196566.796}
SPL {X  -162.820, Y  +671.700, Z    +0.000, E1    -0.272, E3 +196566.137}
SPL {X  -162.820, Y  +669.993, Z    +0.000, E1    +1.755, E3 +196565.804}
SPL {X  -162.820, Y  +666.307, Z    +0.000, E1    +6.851, E3 +196565.691}
SPL {X  -162.820, Y  +660.761, Z    +0.000, E1   +16.102, E3 +196565.834}
SPL {X  -162.820, Y  +655.024, Z    +0.000, E1   +25.730, E3 +196565.995}
SPL {X  -162.820, Y  +646.498, Z    +0.000, E1   +39.738, E3 +196564.516}
SPL {X  -162.820, Y  +637.711, Z    +0.000, E1   +46.793, E3 +196569.008}
SPL {X  -162.820, Y  +598.602, Z    +0.000, E1   +67.541, E3 +196571.559}
SPL {X  -162.820, Y  +578.435, Z    +0.000, E1   +65.472, E3 +196589.659}
SPL {X  -162.820, Y  +475.450, Z    +0.000, E1   +67.130, E3 +196658.597}
ENDSPLINE

SPLINE
SPL {X  -162.820, Y  +483.223, Z    +0.000, E1   +64.312, E3 +196673.036}
SPL {X  -162.820, Y  +502.830, Z    +0.000, E1   +59.229, E3 +196687.957}
ENDSPLINE

SPLINE
SPL {X  -162.820, Y  +486.621, Z    +0.000, E1   +59.661, E3 +196704.877}
SPL {X  -162.820, Y  +472.771, Z    +0.000, E1   +60.369, E3 +196716.622}
SPL {X  -162.820, Y  +460.138, Z    +0.000, E1   +61.014, E3 +196726.942}
SPL {X  -162.820, Y  +448.741, Z    +0.000, E1   +61.510, E3 +196736.456}
SPL {X  -162.820, Y  +430.985, Z    +0.000, E1   +62.533, E3 +196748.889}
SPL {X  -162.820, Y  +413.005, Z    +0.000, E1   +63.234, E3 +196762.879}
SPL {X  -162.820, Y  +396.727, Z    +0.000, E1   +63.972, E3 +196774.231}
SPL {X  -162.756, Y  +375.937, Z    +0.000, E1   +64.914, E3 +196787.840}
SPL {X  -161.353, Y  +358.691, Z    +0.000, E1   +65.588, E3 +196799.065}
SPL {X  -159.475, Y  +347.667, Z    +0.000, E1   +65.889, E3 +196806.945}
SPL {X  -157.043, Y  +337.513, Z    +0.000, E1   +65.541, E3 +196819.023}
SPL {X  -154.736, Y  +329.832, Z    +0.000, E1   +65.034, E3 +196829.469}
SPL {X  -151.631, Y  +321.184, Z    +0.000, E1   +64.776, E3 +196839.314}
SPL {X  -147.832, Y  +312.265, Z    +0.000, E1   +64.201, E3 +196851.123}
SPL {X  -145.264, Y  +306.955, Z    +0.000, E1   +63.555, E3 +196859.729}
SPL {X  -142.454, Y  +301.650, Z    +0.000, E1   +63.360, E3 +196865.733}
SPL {X  -139.696, Y  +296.861, Z    +0.000, E1   +62.910, E3 +196872.501}
SPL {X  -137.330, Y  +293.030, Z    +0.000, E1   +62.290, E3 +196879.126}
SPL {X  -134.245, Y  +288.366, Z    +0.000, E1   +62.031, E3 +196884.607}
SPL {X  -128.642, Y  +280.693, Z    +0.000, E1   +63.351, E3 +196885.601}
SPL {X   -90.696, Y  +245.280, Z    +0.000, E1   +54.124, E3 +197006.289}
ENDSPLINE

SPLINE
SPL {X  -134.058, Y  +288.094, Z    +0.000, E1   +46.503, E3 +197133.803}
SPL {X  -148.633, Y  +314.028, Z    +0.000, E1   +38.752, E3 +197142.692}
SPL {X  -156.325, Y  +334.971, Z    +0.000, E1   +30.037, E3 +197146.460}
SPL {X  -160.130, Y  +351.024, Z    +0.000, E1   +21.715, E3 +197149.774}
SPL {X  -162.127, Y  +365.491, Z    +0.000, E1   +12.692, E3 +197149.697}
SPL {X  -162.801, Y  +378.004, Z    +0.000, E1    +3.811, E3 +197150.113}
SPL {X  -162.820, Y  +382.997, Z    +0.000, E1    -0.389, E3 +197149.437}
SPL {X  -162.820, Y  +387.631, Z    +0.000, E1    -7.169, E3 +197149.196}
SPL {X  -162.820, Y  +394.064, Z    +0.000, E1   -18.298, E3 +197149.007}
SPL {X  -162.820, Y  +402.037, Z    +0.000, E1   -32.247, E3 +197148.928}
SPL {X  -162.820, Y  +414.067, Z    +0.000, E1   -47.235, E3 +197150.354}
SPL {X  -162.820, Y  +424.566, Z    +0.000, E1   -59.255, E3 +197147.020}
SPL {X  -162.820, Y  +460.664, Z    +0.000, E1   -69.605, E3 +197155.316}
SPL {X  -162.820, Y  +481.040, Z    +0.000, E1   -67.047, E3 +197173.904}
SPL {X  -162.820, Y  +573.811, Z    +0.000, E1   -65.269, E3 +197253.647}
SPL {X  -162.820, Y  +580.233, Z    +0.000, E1   -64.427, E3 +197266.353}
SPL {X  -162.820, Y  +590.756, Z    +0.000, E1   -64.410, E3 +197276.921}
SPL {X  -162.820, Y  +600.605, Z    +0.000, E1   -64.446, E3 +197286.494}
SPL {X  -162.820, Y  +611.699, Z    +0.000, E1   -64.369, E3 +197298.174}
SPL {X  -162.820, Y  +622.825, Z    +0.000, E1   -64.446, E3 +197308.618}
SPL {X  -162.820, Y  +635.776, Z    +0.000, E1   -64.495, E3 +197321.308}
SPL {X  -162.820, Y  +648.933, Z    +0.000, E1   -64.417, E3 +197334.855}
SPL {X  -162.820, Y  +658.800, Z    +0.000, E1   -64.418, E3 +197344.669}
SPL {X  -162.820, Y  +670.777, Z    +0.000, E1   -64.432, E3 +197356.582}
SPL {X  -162.296, Y  +686.556, Z    +0.000, E1   -64.388, E3 +197372.786}
SPL {X  -160.469, Y  +701.070, Z    +0.000, E1   -64.058, E3 +197389.689}
SPL {X  -157.811, Y  +713.575, Z    +0.000, E1   -63.758, E3 +197404.267}
SPL {X  -155.696, Y  +721.135, Z    +0.000, E1   -63.387, E3 +197414.201}
SPL {X  -153.915, Y  +726.609, Z    +0.000, E1   -63.196, E3 +197420.975}
SPL {X  -151.802, Y  +732.376, Z    +0.000, E1   -62.761, E3 +197429.517}
SPL {X  -149.758, Y  +737.398, Z    +0.000, E1   -62.434, E3 +197436.537}
SPL {X  -146.903, Y  +743.713, Z    +0.000, E1   -62.188, E3 +197444.310}
SPL {X  -143.515, Y  +750.401, Z    +0.000, E1   -61.484, E3 +197454.994}
SPL {X  -140.303, Y  +756.116, Z    +0.000, E1   -60.974, E3 +197463.192}
SPL {X  -137.124, Y  +761.291, Z    +0.000, E1   -60.398, E3 +197471.239}
SPL {X  -130.896, Y  +770.333, Z    +0.000, E1   -61.755, E3 +197473.913}
SPL {X   -94.739, Y  +805.919, Z    +0.000, E1   -54.063, E3 +197582.230}
ENDSPLINE

SPLINE
SPL {X  -130.051, Y  +771.465, Z    +0.000, E1   -46.832, E3 +197704.014}
SPL {X  -154.243, Y  +725.647, Z    +0.000, E1   -32.659, E3 +197725.576}
SPL {X  -160.324, Y  +701.901, Z    +0.000, E1   -20.534, E3 +197726.399}
SPL {X  -161.938, Y  +690.423, Z    +0.000, E1   -13.625, E3 +197727.789}
SPL {X  -162.638, Y  +681.194, Z    +0.000, E1    -7.430, E3 +197727.610}
SPL {X  -162.820, Y  +672.793, Z    +0.000, E1    -1.263, E3 +197727.668}
SPL {X  -162.820, Y  +670.674, Z    +0.000, E1    +0.808, E3 +197727.199}
SPL {X  -162.820, Y  +666.307, Z    +0.000, E1    +6.851, E3 +197726.981}
SPL {X  -162.820, Y  +660.761, Z    +0.000, E1   +16.102, E3 +197727.124}
SPL {X  -162.820, Y  +655.024, Z    +0.000, E1   +25.730, E3 +197727.285}
SPL {X  -162.820, Y  +646.498, Z    +0.000, E1   +39.738, E3 +197725.806}
SPL {X  -162.820, Y  +637.711, Z    +0.000, E1   +46.793, E3 +197730.299}
SPL {X  -162.820, Y  +598.602, Z    +0.000, E1   +67.541, E3 +197732.850}
SPL {X  -162.820, Y  +578.435, Z    +0.000, E1   +65.472, E3 +197750.949}
SPL {X  -162.820, Y  +475.450, Z    +0.000, E1   +67.130, E3 +197819.887}
ENDSPLINE

SPLINE
SPL {X  -162.820, Y  +483.223, Z    +0.000, E1   +64.312, E3 +197834.326}
SPL {X  -162.820, Y  +502.830, Z    +0.000, E1   +59.229, E3 +197849.247}
ENDSPLINE

SPLINE
SPL {X  -162.820, Y  +486.621, Z    +0.000, E1   +59.661, E3 +197866.167}
SPL {X  -162.820, Y  +472.771, Z    +0.000, E1   +60.369, E3 +197877.912}
SPL {X  -162.820, Y  +460.138, Z    +0.000, E1   +61.014, E3 +197888.232}
SPL {X  -162.820, Y  +448.741, Z    +0.000, E1   +61.510, E3 +197897.747}
SPL {X  -162.820, Y  +430.985, Z    +0.000, E1   +62.533, E3 +197910.180}
SPL {X  -162.820, Y  +413.005, Z    +0.000, E1   +63.234, E3 +197924.170}
SPL {X  -162.820, Y  +396.727, Z    +0.000, E1   +63.972, E3 +197935.521}
SPL {X  -162.820, Y  +382.966, Z    +0.000, E1   +64.511, E3 +197945.243}
SPL {X  -161.867, Y  +362.911, Z    +0.000, E1   +65.480, E3 +197957.317}
SPL {X  -159.475, Y  +347.667, Z    +0.000, E1   +65.889, E3 +197968.236}
SPL {X  -157.043, Y  +337.513, Z    +0.000, E1   +65.541, E3 +197980.313}
SPL {X  -153.776, Y  +326.991, Z    +0.000, E1   +65.023, E3 +197993.554}
SPL {X  -149.992, Y  +317.154, Z    +0.000, E1   +64.515, E3 +198006.018}
SPL {X  -146.026, Y  +308.480, Z    +0.000, E1   +63.813, E3 +198018.260}
SPL {X  -142.454, Y  +301.650, Z    +0.000, E1   +63.360, E3 +198027.023}
SPL {X  -139.696, Y  +296.861, Z    +0.000, E1   +62.910, E3 +198033.791}
SPL {X  -137.330, Y  +293.030, Z    +0.000, E1   +62.290, E3 +198040.416}
SPL {X  -134.245, Y  +288.366, Z    +0.000, E1   +62.031, E3 +198045.898}
SPL {X  -128.642, Y  +280.693, Z    +0.000, E1   +63.351, E3 +198046.891}
SPL {X   -90.696, Y  +245.280, Z    +0.000, E1   +54.124, E3 +198167.580}
ENDSPLINE

